LIN {X 0,Y 524.296,Z 355.631,A -85,B 0,C 180,E1 -4781.013,E2 -4781.013} C_VEL
LIN {X 0,Y 524.616,Z 343.771,A -85,B 0,C 180,E1 -4781.889,E2 -4781.889} C_VEL
LIN {X 0,Y 524.905,Z 331.9,A -85,B 0,C 180,E1 -4782.567,E2 -4782.567} C_VEL
LIN {X 0,Y 525.166,Z 319.528,A -85,B 0,C 180,E1 -4783.101,E2 -4783.101} C_VEL
LIN {X 0,Y 525.422,Z 306.835,A -85,B 0,C 180,E1 -4783.489,E2 -4783.489} C_VEL
LIN {X 0,Y 525.58,Z 293.563,A -85,B 0,C 180,E1 -4783.731,E2 -4783.731} C_VEL
LIN {X 0,Y 525.785,Z 203.396,A -85,B 0,C 180,E1 -4784.97,E2 -4784.97} C_VEL
LIN {X 0,Y 524.208,Z 192.625,A -85,B 0,C 180,E1 -4785.178,E2 -4785.178} C_VEL
LIN {X 0,Y 524.604,Z 173.678,A -85,B 0,C 180,E1 -4787.978,E2 -4787.978} C_VEL
LIN {X 0,Y 525.138,Z 150.917,A -85,B 0,C 180,E1 -4791.389,E2 -4791.389} C_VEL
LIN {X 0,Y 525.407,Z 136.058,A -85,B 0,C 180,E1 -4793.659,E2 -4793.659} C_VEL
LIN {X 0,Y 523.975,Z 128.216,A -85,B 0,C 180,E1 -4794.967,E2 -4794.967} C_VEL
LIN {X 0,Y 523.922,Z 128.227,A -85,B 0,C 180,E1 -4798.002,E2 -4798.002} C_VEL
LIN {X 0,Y 523.941,Z 128.22,A -85,B 0,C 180,E1 -4800.854,E2 -4800.854} C_VEL
LIN {X 0,Y 523.962,Z 128.222,A -85,B 0,C 180,E1 -4803.734,E2 -4803.734} C_VEL
LIN {X 0,Y 523.901,Z 128.222,A -85,B 0,C 180,E1 -4806.401,E2 -4806.401} C_VEL
LIN {X 0,Y 523.922,Z 128.22,A -85,B 0,C 180,E1 -4809.085,E2 -4809.085} C_VEL
LIN {X 0,Y 523.942,Z 128.217,A -85,B 0,C 180,E1 -4812.12,E2 -4812.12} C_VEL
LIN {X 0,Y 523.939,Z 128.224,A -85,B 0,C 180,E1 -4815.311,E2 -4815.311} C_VEL
LIN {X 0,Y 523.94,Z 128.218,A -85,B 0,C 180,E1 -4818.692,E2 -4818.692} C_VEL
LIN {X 0,Y 523.914,Z 128.221,A -85,B 0,C 180,E1 -4821.898,E2 -4821.898} C_VEL
LIN {X 0,Y 523.922,Z 128.225,A -85,B 0,C 180,E1 -4824.912,E2 -4824.912} C_VEL
LIN {X 0,Y 523.931,Z 128.219,A -85,B 0,C 180,E1 -4827.681,E2 -4827.681} C_VEL
LIN {X 0,Y 523.935,Z 128.222,A -85,B 0,C 180,E1 -4830.68,E2 -4830.68} C_VEL
LIN {X 0,Y 523.902,Z 128.221,A -85,B 0,C 180,E1 -4833.725,E2 -4833.725} C_VEL
LIN {X 0,Y 523.904,Z 128.223,A -85,B 0,C 180,E1 -4836.269,E2 -4836.269} C_VEL
LIN {X 0,Y 523.928,Z 128.223,A -85,B 0,C 180,E1 -4838.766,E2 -4838.766} C_VEL
LIN {X 0,Y 523.924,Z 128.218,A -85,B 0,C 180,E1 -4841.22,E2 -4841.22} C_VEL
LIN {X 0,Y 523.877,Z 128.224,A -85,B 0,C 180,E1 -4843.637,E2 -4843.637} C_VEL
LIN {X 0,Y 523.959,Z 128.211,A -85,B 0,C 180,E1 -4845.235,E2 -4845.235} C_VEL
LIN {X 0,Y 523.958,Z 128.221,A -85,B 0,C 180,E1 -4848.393,E2 -4848.393} C_VEL
LIN {X 0,Y 523.94,Z 128.214,A -85,B 0,C 180,E1 -4851.515,E2 -4851.515} C_VEL
LIN {X 0,Y 523.997,Z 128.213,A -85,B 0,C 180,E1 -4853.84,E2 -4853.84} C_VEL
LIN {X 0,Y 524.101,Z 128.197,A -85,B 0,C 180,E1 -4857.695,E2 -4857.695} C_VEL
LIN {X 0,Y 524.094,Z 128.204,A -85,B 0,C 180,E1 -4860,E2 -4860} C_VEL
LIN {X 0,Y 524.102,Z 128.195,A -85,B 0,C 180,E1 -4862.306,E2 -4862.306} C_VEL
LIN {X 0,Y 524,Z 128.211,A -85,B 0,C 180,E1 -4866.16,E2 -4866.16} C_VEL
LIN {X 0,Y 523.977,Z 128.212,A -85,B 0,C 180,E1 -4869.262,E2 -4869.262} C_VEL
LIN {X 0,Y 523.997,Z 128.214,A -85,B 0,C 180,E1 -4871.736,E2 -4871.736} C_VEL
LIN {X 0,Y 523.983,Z 128.212,A -85,B 0,C 180,E1 -4875.048,E2 -4875.048} C_VEL
LIN {X 0,Y 523.944,Z 128.216,A -85,B 0,C 180,E1 -4877.97,E2 -4877.97} C_VEL
LIN {X 0,Y 523.958,Z 128.213,A -85,B 0,C 180,E1 -4880.411,E2 -4880.411} C_VEL
LIN {X 0,Y 523.907,Z 128.226,A -85,B 0,C 180,E1 -4882.894,E2 -4882.894} C_VEL
LIN {X 0,Y 523.903,Z 128.224,A -85,B 0,C 180,E1 -4885.421,E2 -4885.421} C_VEL
LIN {X 0,Y 523.92,Z 128.218,A -85,B 0,C 180,E1 -4888.002,E2 -4888.002} C_VEL
LIN {X 0,Y 523.936,Z 128.225,A -85,B 0,C 180,E1 -4890.853,E2 -4890.853} C_VEL
LIN {X 0,Y 523.931,Z 128.217,A -85,B 0,C 180,E1 -4893.73,E2 -4893.73} C_VEL
LIN {X 0,Y 523.905,Z 128.225,A -85,B 0,C 180,E1 -4896.401,E2 -4896.401} C_VEL
LIN {X 0,Y 523.915,Z 128.22,A -85,B 0,C 180,E1 -4899.086,E2 -4899.086} C_VEL
LIN {X 0,Y 523.953,Z 128.214,A -85,B 0,C 180,E1 -4902.119,E2 -4902.119} C_VEL
LIN {X 0,Y 523.946,Z 128.215,A -85,B 0,C 180,E1 -4905.31,E2 -4905.31} C_VEL
LIN {X 0,Y 523.904,Z 128.222,A -85,B 0,C 180,E1 -4906.869,E2 -4906.869} C_VEL
LIN {X 0,Y 523.232,Z 128.305,A -85,B 0,C 180,E1 -4907.51,E2 -4907.51} C_VEL
LIN {X 0,Y 520.37,Z 128.666,A -85,B 0,C 180,E1 -4908.552,E2 -4908.552} C_VEL
LIN {X 0,Y 517.967,Z 128.963,A -85,B 0,C 180,E1 -4909.391,E2 -4909.391} C_VEL
LIN {X 0,Y 516.956,Z 129.093,A -85,B 0,C 180,E1 -4910.039,E2 -4910.039} C_VEL
LIN {X 0,Y 516.885,Z 129.102,A -85,B 0,C 180,E1 -4910.258,E2 -4910.258} C_VEL
LIN {X 0,Y 516.881,Z 129.097,A -85,B 0,C 180,E1 -4913.343,E2 -4913.343} C_VEL
LIN {X 0,Y 516.911,Z 129.099,A -85,B 0,C 180,E1 -4916.121,E2 -4916.121} C_VEL
LIN {X 0,Y 516.896,Z 129.095,A -85,B 0,C 180,E1 -4918.936,E2 -4918.936} C_VEL
LIN {X 0,Y 516.914,Z 129.099,A -85,B 0,C 180,E1 -4921.584,E2 -4921.584} C_VEL
LIN {X 0,Y 516.937,Z 129.095,A -85,B 0,C 180,E1 -4924.211,E2 -4924.211} C_VEL
LIN {X 0,Y 516.978,Z 129.251,A -85,B 0,C 180,E1 -4925.931,E2 -4925.931} C_VEL
LIN {X 0,Y 517.464,Z 133.566,A -85,B 0,C 180,E1 -4926.804,E2 -4926.804} C_VEL
LIN {X 0,Y 517.266,Z 148.39,A -85,B 0,C 180,E1 -4929.687,E2 -4929.687} C_VEL
LIN {X 0,Y 519.159,Z 158.865,A -85,B 0,C 180,E1 -4929.9,E2 -4929.9} C_VEL
LIN {X 0,Y 518.678,Z 255.148,A -85,B 0,C 180,E1 -4931.256,E2 -4931.256} C_VEL
LIN {X 0,Y 518.464,Z 268.883,A -85,B 0,C 180,E1 -4931.617,E2 -4931.617} C_VEL
LIN {X 0,Y 518.279,Z 280.763,A -85,B 0,C 180,E1 -4932.082,E2 -4932.082} C_VEL
LIN {X 0,Y 518.008,Z 293.082,A -85,B 0,C 180,E1 -4932.735,E2 -4932.735} C_VEL
LIN {X 0,Y 517.682,Z 304.709,A -85,B 0,C 180,E1 -4933.536,E2 -4933.536} C_VEL
LIN {X 0,Y 517.386,Z 314.85,A -85,B 0,C 180,E1 -4934.411,E2 -4934.411} C_VEL
LIN {X 0,Y 517.145,Z 324.44,A -85,B 0,C 180,E1 -4935.438,E2 -4935.438} C_VEL
LIN {X 0,Y 516.818,Z 333.435,A -85,B 0,C 180,E1 -4936.633,E2 -4936.633} C_VEL
LIN {X 0,Y 516.649,Z 340.641,A -85,B 0,C 180,E1 -4937.827,E2 -4937.827} C_VEL
LIN {X 0,Y 516.461,Z 346.349,A -85,B 0,C 180,E1 -4939.017,E2 -4939.017} C_VEL
LIN {X 0,Y 516.384,Z 350.822,A -85,B 0,C 180,E1 -4940.204,E2 -4940.204} C_VEL
LIN {X 0,Y 516.348,Z 354.202,A -85,B 0,C 180,E1 -4941.389,E2 -4941.389} C_VEL
LIN {X 0,Y 516.292,Z 357.143,A -85,B 0,C 180,E1 -4942.962,E2 -4942.962} C_VEL
LIN {X 0,Y 516.313,Z 358.016,A -85,B 0,C 180,E1 -4943.748,E2 -4943.748} C_VEL
LIN {X 0,Y 516.309,Z 358.461,A -85,B 0,C 180,E1 -4944.532,E2 -4944.532} C_VEL
LIN {X 0,Y 516.326,Z 358.176,A -85,B 0,C 180,E1 -4946.097,E2 -4946.097} C_VEL
LIN {X 0,Y 516.344,Z 357.465,A -85,B 0,C 180,E1 -4946.878,E2 -4946.878} C_VEL
LIN {X 0,Y 516.267,Z 356.334,A -85,B 0,C 180,E1 -4947.659,E2 -4947.659} C_VEL
LIN {X 0,Y 516.253,Z 352.833,A -85,B 0,C 180,E1 -4949.219,E2 -4949.219} C_VEL
LIN {X 0,Y 516.445,Z 349.035,A -85,B 0,C 180,E1 -4950.389,E2 -4950.389} C_VEL
LIN {X 0,Y 516.44,Z 344.15,A -85,B 0,C 180,E1 -4951.559,E2 -4951.559} C_VEL
LIN {X 0,Y 516.671,Z 338.002,A -85,B 0,C 180,E1 -4952.728,E2 -4952.728} C_VEL
LIN {X 0,Y 516.803,Z 330.352,A -85,B 0,C 180,E1 -4953.898,E2 -4953.898} C_VEL
LIN {X 0,Y 517.111,Z 322.535,A -85,B 0,C 180,E1 -4954.872,E2 -4954.872} C_VEL
LIN {X 0,Y 517.454,Z 311.966,A -85,B 0,C 180,E1 -4955.944,E2 -4955.944} C_VEL
LIN {X 0,Y 517.824,Z 301.13,A -85,B 0,C 180,E1 -4956.82,E2 -4956.82} C_VEL
LIN {X 0,Y 518.163,Z 289.248,A -85,B 0,C 180,E1 -4957.573,E2 -4957.573} C_VEL
LIN {X 0,Y 518.355,Z 277.548,A -85,B 0,C 180,E1 -4958.147,E2 -4958.147} C_VEL
LIN {X 0,Y 518.562,Z 264.854,A -85,B 0,C 180,E1 -4958.597,E2 -4958.597} C_VEL
LIN {X 0,Y 518.631,Z 251.952,A -85,B 0,C 180,E1 -4958.891,E2 -4958.891} C_VEL
LIN {X 0,Y 519.083,Z 157.954,A -85,B 0,C 180,E1 -4960.204,E2 -4960.204} C_VEL
LIN {X 0,Y 517.203,Z 148.275,A -85,B 0,C 180,E1 -4960.421,E2 -4960.421} C_VEL
LIN {X 0,Y 517.436,Z 133.231,A -85,B 0,C 180,E1 -4963.349,E2 -4963.349} C_VEL
LIN {X 0,Y 516.945,Z 129.096,A -85,B 0,C 180,E1 -4964.214,E2 -4964.214} C_VEL
LIN {X 0,Y 516.907,Z 129.094,A -85,B 0,C 180,E1 -4967.404,E2 -4967.404} C_VEL
LIN {X 0,Y 516.94,Z 129.097,A -85,B 0,C 180,E1 -4970.267,E2 -4970.267} C_VEL
LIN {X 0,Y 516.86,Z 129.098,A -85,B 0,C 180,E1 -4973.223,E2 -4973.223} C_VEL
LIN {X 0,Y 516.941,Z 129.095,A -85,B 0,C 180,E1 -4976.195,E2 -4976.195} C_VEL
LIN {X 0,Y 516.919,Z 129.092,A -85,B 0,C 180,E1 -4979.303,E2 -4979.303} C_VEL
LIN {X 0,Y 516.893,Z 129.096,A -85,B 0,C 180,E1 -4982.542,E2 -4982.542} C_VEL
LIN {X 0,Y 516.863,Z 129.101,A -85,B 0,C 180,E1 -4985.328,E2 -4985.328} C_VEL
LIN {X 0,Y 516.876,Z 129.102,A -85,B 0,C 180,E1 -4987.942,E2 -4987.942} C_VEL
LIN {X 0,Y 516.878,Z 129.097,A -85,B 0,C 180,E1 -4990.741,E2 -4990.741} C_VEL
LIN {X 0,Y 516.877,Z 129.098,A -85,B 0,C 180,E1 -4992.83,E2 -4992.83} C_VEL
LIN {X 0,Y 516.889,Z 129.099,A -85,B 0,C 180,E1 -4995.006,E2 -4995.006} C_VEL
LIN {X 0,Y 516.906,Z 129.094,A -85,B 0,C 180,E1 -4998.398,E2 -4998.398} C_VEL
LIN {X 0,Y 516.871,Z 129.104,A -85,B 0,C 180,E1 -5001.283,E2 -5001.283} C_VEL
LIN {X 0,Y 516.862,Z 129.099,A -85,B 0,C 180,E1 -5004.219,E2 -5004.219} C_VEL
LIN {X 0,Y 516.872,Z 129.103,A -85,B 0,C 180,E1 -5007.051,E2 -5007.051} C_VEL
LIN {X 0,Y 516.876,Z 129.098,A -85,B 0,C 180,E1 -5009.795,E2 -5009.795} C_VEL
LIN {X 0,Y 516.91,Z 129.097,A -85,B 0,C 180,E1 -5012.466,E2 -5012.466} C_VEL
LIN {X 0,Y 516.861,Z 129.1,A -85,B 0,C 180,E1 -5015.645,E2 -5015.645} C_VEL
LIN {X 0,Y 516.873,Z 129.103,A -85,B 0,C 180,E1 -5018.461,E2 -5018.461} C_VEL
LIN {X 0,Y 516.878,Z 129.102,A -85,B 0,C 180,E1 -5020.954,E2 -5020.954} C_VEL
LIN {X 0,Y 516.86,Z 129.1,A -85,B 0,C 180,E1 -5023.408,E2 -5023.408} C_VEL
LIN {X 0,Y 516.86,Z 129.101,A -85,B 0,C 180,E1 -5025.833,E2 -5025.833} C_VEL
LIN {X 0,Y 516.935,Z 129.092,A -85,B 0,C 180,E1 -5029.027,E2 -5029.027} C_VEL
LIN {X 0,Y 516.929,Z 129.096,A -85,B 0,C 180,E1 -5032.186,E2 -5032.186} C_VEL
LIN {X 0,Y 516.972,Z 129.09,A -85,B 0,C 180,E1 -5034.539,E2 -5034.539} C_VEL
LIN {X 0,Y 517.061,Z 129.078,A -85,B 0,C 180,E1 -5037.663,E2 -5037.663} C_VEL
LIN {X 0,Y 517.052,Z 129.081,A -85,B 0,C 180,E1 -5040,E2 -5040} C_VEL
LIN {X 0,Y 517.061,Z 129.078,A -85,B 0,C 180,E1 -5042.337,E2 -5042.337} C_VEL
LIN {X 0,Y 516.972,Z 129.089,A -85,B 0,C 180,E1 -5046.244,E2 -5046.244} C_VEL
LIN {X 0,Y 516.923,Z 129.097,A -85,B 0,C 180,E1 -5049.39,E2 -5049.39} C_VEL
LIN {X 0,Y 516.939,Z 129.094,A -85,B 0,C 180,E1 -5051.807,E2 -5051.807} C_VEL
LIN {X 0,Y 516.923,Z 129.096,A -85,B 0,C 180,E1 -5055.143,E2 -5055.143} C_VEL
LIN {X 0,Y 516.899,Z 129.095,A -85,B 0,C 180,E1 -5058.223,E2 -5058.223} C_VEL
LIN {X 0,Y 516.892,Z 129.097,A -85,B 0,C 180,E1 -5060.702,E2 -5060.702} C_VEL
LIN {X 0,Y 516.872,Z 129.098,A -85,B 0,C 180,E1 -5064.074,E2 -5064.074} C_VEL
LIN {X 0,Y 516.896,Z 129.098,A -85,B 0,C 180,E1 -5066.659,E2 -5066.659} C_VEL
LIN {X 0,Y 516.898,Z 129.097,A -85,B 0,C 180,E1 -5069.524,E2 -5069.524} C_VEL
LIN {X 0,Y 516.884,Z 129.1,A -85,B 0,C 180,E1 -5072.544,E2 -5072.544} C_VEL
LIN {X 0,Y 516.856,Z 129.102,A -85,B 0,C 180,E1 -5075.33,E2 -5075.33} C_VEL
LIN {X 0,Y 516.871,Z 129.098,A -85,B 0,C 180,E1 -5077.944,E2 -5077.944} C_VEL
LIN {X 0,Y 516.874,Z 129.103,A -85,B 0,C 180,E1 -5080.743,E2 -5080.743} C_VEL
LIN {X 0,Y 516.875,Z 129.101,A -85,B 0,C 180,E1 -5082.832,E2 -5082.832} C_VEL
LIN {X 0,Y 516.888,Z 129.098,A -85,B 0,C 180,E1 -5085.008,E2 -5085.008} C_VEL
LIN {X 0,Y 516.907,Z 129.1,A -85,B 0,C 180,E1 -5088.4,E2 -5088.4} C_VEL
LIN {X 0,Y 516.876,Z 129.097,A -85,B 0,C 180,E1 -5091.285,E2 -5091.285} C_VEL
LIN {X 0,Y 516.866,Z 129.105,A -85,B 0,C 180,E1 -5094.221,E2 -5094.221} C_VEL
LIN {X 0,Y 516.891,Z 129.095,A -85,B 0,C 180,E1 -5097.054,E2 -5097.054} C_VEL
LIN {X 0,Y 516.889,Z 129.1,A -85,B 0,C 180,E1 -5099.797,E2 -5099.797} C_VEL
LIN {X 0,Y 516.925,Z 129.093,A -85,B 0,C 180,E1 -5102.468,E2 -5102.468} C_VEL
LIN {X 0,Y 516.953,Z 129.223,A -85,B 0,C 180,E1 -5104.941,E2 -5104.941} C_VEL
LIN {X 0,Y 518.403,Z 136.998,A -85,B 0,C 180,E1 -5106.215,E2 -5106.215} C_VEL
LIN {X 0,Y 518.207,Z 149.253,A -85,B 0,C 180,E1 -5108.103,E2 -5108.103} C_VEL
LIN {X 0,Y 517.782,Z 165.52,A -85,B 0,C 180,E1 -5110.578,E2 -5110.578} C_VEL
LIN {X 0,Y 517.435,Z 184.423,A -85,B 0,C 180,E1 -5113.428,E2 -5113.428} C_VEL
LIN {X 0,Y 517.213,Z 192.423,A -85,B 0,C 180,E1 -5114.625,E2 -5114.625} C_VEL
LIN {X 0,Y 519.016,Z 205.194,A -85,B 0,C 180,E1 -5114.86,E2 -5114.86} C_VEL
LIN {X 0,Y 518.594,Z 301.016,A -85,B 0,C 180,E1 -5116.207,E2 -5116.207} C_VEL
LIN {X 0,Y 518.375,Z 313.548,A -85,B 0,C 180,E1 -5116.526,E2 -5116.526} C_VEL
LIN {X 0,Y 518.073,Z 326.498,A -85,B 0,C 180,E1 -5117.017,E2 -5117.017} C_VEL
LIN {X 0,Y 517.775,Z 338.996,A -85,B 0,C 180,E1 -5117.669,E2 -5117.669} C_VEL
LIN {X 0,Y 517.478,Z 350.426,A -85,B 0,C 180,E1 -5118.445,E2 -5118.445} C_VEL
LIN {X 0,Y 517.194,Z 360.897,A -85,B 0,C 180,E1 -5119.331,E2 -5119.331} C_VEL
LIN {X 0,Y 516.905,Z 369.459,A -85,B 0,C 180,E1 -5120.216,E2 -5120.216} C_VEL
LIN {X 0,Y 516.68,Z 377.362,A -85,B 0,C 180,E1 -5121.199,E2 -5121.199} C_VEL
LIN {X 0,Y 516.515,Z 385.085,A -85,B 0,C 180,E1 -5122.377,E2 -5122.377} C_VEL
LIN {X 0,Y 516.373,Z 392.205,A -85,B 0,C 180,E1 -5123.75,E2 -5123.75} C_VEL
LIN {X 0,Y 516.312,Z 396.943,A -85,B 0,C 180,E1 -5124.925,E2 -5124.925} C_VEL
LIN {X 0,Y 516.351,Z 400.566,A -85,B 0,C 180,E1 -5126.099,E2 -5126.099} C_VEL
LIN {X 0,Y 516.303,Z 402.432,A -85,B 0,C 180,E1 -5126.88,E2 -5126.88} C_VEL
LIN {X 0,Y 516.264,Z 403.831,A -85,B 0,C 180,E1 -5127.66,E2 -5127.66} C_VEL
LIN {X 0,Y 516.172,Z 405.435,A -85,B 0,C 180,E1 -5129.221,E2 -5129.221} C_VEL
LIN {X 0,Y 516.173,Z 405.651,A -85,B 0,C 180,E1 -5130.001,E2 -5130.001} C_VEL
LIN {X 0,Y 516.193,Z 404.822,A -85,B 0,C 180,E1 -5131.561,E2 -5131.561} C_VEL
LIN {X 0,Y 516.264,Z 403.825,A -85,B 0,C 180,E1 -5132.341,E2 -5132.341} C_VEL
LIN {X 0,Y 516.303,Z 402.425,A -85,B 0,C 180,E1 -5133.122,E2 -5133.122} C_VEL
LIN {X 0,Y 516.31,Z 399.476,A -85,B 0,C 180,E1 -5134.294,E2 -5134.294} C_VEL
LIN {X 0,Y 516.367,Z 395.487,A -85,B 0,C 180,E1 -5135.468,E2 -5135.468} C_VEL
LIN {X 0,Y 516.427,Z 389.342,A -85,B 0,C 180,E1 -5136.841,E2 -5136.841} C_VEL
LIN {X 0,Y 516.568,Z 382.649,A -85,B 0,C 180,E1 -5138.017,E2 -5138.017} C_VEL
LIN {X 0,Y 516.756,Z 374.336,A -85,B 0,C 180,E1 -5139.196,E2 -5139.196} C_VEL
LIN {X 0,Y 516.985,Z 365.819,A -85,B 0,C 180,E1 -5140.18,E2 -5140.18} C_VEL
LIN {X 0,Y 517.302,Z 355.3,A -85,B 0,C 180,E1 -5141.163,E2 -5141.163} C_VEL
LIN {X 0,Y 517.623,Z 343.438,A -85,B 0,C 180,E1 -5142.052,E2 -5142.052} C_VEL
LIN {X 0,Y 517.941,Z 331.566,A -85,B 0,C 180,E1 -5142.739,E2 -5142.739} C_VEL
LIN {X 0,Y 518.227,Z 319.193,A -85,B 0,C 180,E1 -5143.28,E2 -5143.28} C_VEL
LIN {X 0,Y 518.506,Z 306.499,A -85,B 0,C 180,E1 -5143.672,E2 -5143.672} C_VEL
LIN {X 0,Y 518.675,Z 291.432,A -85,B 0,C 180,E1 -5143.942,E2 -5143.942} C_VEL
LIN {X 0,Y 518.91,Z 204.051,A -85,B 0,C 180,E1 -5145.159,E2 -5145.159} C_VEL
LIN {X 0,Y 517.223,Z 192.309,A -85,B 0,C 180,E1 -5145.386,E2 -5145.386} C_VEL
LIN {X 0,Y 517.725,Z 170.878,A -85,B 0,C 180,E1 -5148.603,E2 -5148.603} C_VEL
LIN {X 0,Y 518.192,Z 152,A -85,B 0,C 180,E1 -5151.481,E2 -5151.481} C_VEL
LIN {X 0,Y 518.466,Z 137.166,A -85,B 0,C 180,E1 -5153.783,E2 -5153.783} C_VEL
LIN {X 0,Y 516.916,Z 129.095,A -85,B 0,C 180,E1 -5155.143,E2 -5155.143} C_VEL
LIN {X 0,Y 516.886,Z 129.103,A -85,B 0,C 180,E1 -5157.896,E2 -5157.896} C_VEL
LIN {X 0,Y 516.889,Z 129.104,A -85,B 0,C 180,E1 -5160.204,E2 -5160.204} C_VEL
LIN {X 0,Y 516.898,Z 129.096,A -85,B 0,C 180,E1 -5162.947,E2 -5162.947} C_VEL
LIN {X 0,Y 516.87,Z 129.105,A -85,B 0,C 180,E1 -5165.781,E2 -5165.781} C_VEL
LIN {X 0,Y 516.882,Z 129.095,A -85,B 0,C 180,E1 -5168.716,E2 -5168.716} C_VEL
LIN {X 0,Y 516.907,Z 129.097,A -85,B 0,C 180,E1 -5171.776,E2 -5171.776} C_VEL
LIN {X 0,Y 516.897,Z 129.097,A -85,B 0,C 180,E1 -5175.007,E2 -5175.007} C_VEL
LIN {X 0,Y 516.903,Z 129.093,A -85,B 0,C 180,E1 -5178.4,E2 -5178.4} C_VEL
LIN {X 0,Y 516.877,Z 129.104,A -85,B 0,C 180,E1 -5181.284,E2 -5181.284} C_VEL
LIN {X 0,Y 516.868,Z 129.098,A -85,B 0,C 180,E1 -5184.219,E2 -5184.219} C_VEL
LIN {X 0,Y 516.88,Z 129.104,A -85,B 0,C 180,E1 -5187.052,E2 -5187.052} C_VEL
LIN {X 0,Y 516.862,Z 129.098,A -85,B 0,C 180,E1 -5189.794,E2 -5189.794} C_VEL
LIN {X 0,Y 516.874,Z 129.099,A -85,B 0,C 180,E1 -5192.464,E2 -5192.464} C_VEL
LIN {X 0,Y 516.844,Z 129.105,A -85,B 0,C 180,E1 -5195.068,E2 -5195.068} C_VEL
LIN {X 0,Y 516.869,Z 129.097,A -85,B 0,C 180,E1 -5197.622,E2 -5197.622} C_VEL
LIN {X 0,Y 516.913,Z 129.092,A -85,B 0,C 180,E1 -5200.129,E2 -5200.129} C_VEL
LIN {X 0,Y 516.877,Z 129.103,A -85,B 0,C 180,E1 -5202.594,E2 -5202.594} C_VEL
LIN {X 0,Y 516.929,Z 129.088,A -85,B 0,C 180,E1 -5205.03,E2 -5205.03} C_VEL
LIN {X 0,Y 516.918,Z 129.098,A -85,B 0,C 180,E1 -5208.233,E2 -5208.233} C_VEL
LIN {X 0,Y 516.914,Z 129.088,A -85,B 0,C 180,E1 -5211.399,E2 -5211.399} C_VEL
LIN {X 0,Y 516.975,Z 129.086,A -85,B 0,C 180,E1 -5214.539,E2 -5214.539} C_VEL
LIN {X 0,Y 517.07,Z 129.073,A -85,B 0,C 180,E1 -5217.663,E2 -5217.663} C_VEL
LIN {X 0,Y 517.063,Z 129.08,A -85,B 0,C 180,E1 -5220,E2 -5220} C_VEL
LIN {X 0,Y 517.071,Z 129.07,A -85,B 0,C 180,E1 -5222.337,E2 -5222.337} C_VEL
LIN {X 0,Y 516.967,Z 129.086,A -85,B 0,C 180,E1 -5226.244,E2 -5226.244} C_VEL
LIN {X 0,Y 516.934,Z 129.091,A -85,B 0,C 180,E1 -5229.39,E2 -5229.39} C_VEL
LIN {X 0,Y 516.952,Z 129.091,A -85,B 0,C 180,E1 -5231.807,E2 -5231.807} C_VEL
LIN {X 0,Y 516.936,Z 129.091,A -85,B 0,C 180,E1 -5235.143,E2 -5235.143} C_VEL
LIN {X 0,Y 516.911,Z 129.091,A -85,B 0,C 180,E1 -5238.223,E2 -5238.223} C_VEL
LIN {X 0,Y 516.905,Z 129.093,A -85,B 0,C 180,E1 -5240.702,E2 -5240.702} C_VEL
LIN {X 0,Y 516.885,Z 129.093,A -85,B 0,C 180,E1 -5244.074,E2 -5244.074} C_VEL
LIN {X 0,Y 516.895,Z 129.098,A -85,B 0,C 180,E1 -5246.66,E2 -5246.66} C_VEL
LIN {X 0,Y 516.908,Z 129.093,A -85,B 0,C 180,E1 -5249.523,E2 -5249.523} C_VEL
LIN {X 0,Y 516.895,Z 129.099,A -85,B 0,C 180,E1 -5252.543,E2 -5252.543} C_VEL
LIN {X 0,Y 516.867,Z 129.098,A -85,B 0,C 180,E1 -5255.33,E2 -5255.33} C_VEL
LIN {X 0,Y 516.881,Z 129.096,A -85,B 0,C 180,E1 -5257.943,E2 -5257.943} C_VEL
LIN {X 0,Y 516.885,Z 129.094,A -85,B 0,C 180,E1 -5260.742,E2 -5260.742} C_VEL
LIN {X 0,Y 516.885,Z 129.098,A -85,B 0,C 180,E1 -5262.832,E2 -5262.832} C_VEL
LIN {X 0,Y 516.898,Z 129.094,A -85,B 0,C 180,E1 -5265.007,E2 -5265.007} C_VEL
LIN {X 0,Y 516.913,Z 129.098,A -85,B 0,C 180,E1 -5268.399,E2 -5268.399} C_VEL
LIN {X 0,Y 516.885,Z 129.102,A -85,B 0,C 180,E1 -5270.258,E2 -5270.258} C_VEL
LIN {X 0,Y 516.249,Z 129.188,A -85,B 0,C 180,E1 -5270.908,E2 -5270.908} C_VEL
LIN {X 0,Y 513.406,Z 129.544,A -85,B 0,C 180,E1 -5271.963,E2 -5271.963} C_VEL
LIN {X 0,Y 510.976,Z 129.841,A -85,B 0,C 180,E1 -5272.813,E2 -5272.813} C_VEL
LIN {X 0,Y 509.918,Z 129.968,A -85,B 0,C 180,E1 -5273.47,E2 -5273.47} C_VEL
LIN {X 0,Y 509.826,Z 129.978,A -85,B 0,C 180,E1 -5273.692,E2 -5273.692} C_VEL
LIN {X 0,Y 509.863,Z 129.972,A -85,B 0,C 180,E1 -5276.539,E2 -5276.539} C_VEL
LIN {X 0,Y 509.85,Z 129.974,A -85,B 0,C 180,E1 -5279.334,E2 -5279.334} C_VEL
LIN {X 0,Y 509.888,Z 129.974,A -85,B 0,C 180,E1 -5282.054,E2 -5282.054} C_VEL
LIN {X 0,Y 509.884,Z 129.971,A -85,B 0,C 180,E1 -5284.704,E2 -5284.704} C_VEL
LIN {X 0,Y 509.925,Z 130.125,A -85,B 0,C 180,E1 -5285.793,E2 -5285.793} C_VEL
LIN {X 0,Y 510.486,Z 134.461,A -85,B 0,C 180,E1 -5286.683,E2 -5286.683} C_VEL
LIN {X 0,Y 510.303,Z 148.728,A -85,B 0,C 180,E1 -5289.474,E2 -5289.474} C_VEL
LIN {X 0,Y 512.299,Z 159.889,A -85,B 0,C 180,E1 -5289.7,E2 -5289.7} C_VEL
LIN {X 0,Y 511.813,Z 255.635,A -85,B 0,C 180,E1 -5291.07,E2 -5291.07} C_VEL
LIN {X 0,Y 511.577,Z 269.311,A -85,B 0,C 180,E1 -5291.435,E2 -5291.435} C_VEL
LIN {X 0,Y 511.364,Z 281.795,A -85,B 0,C 180,E1 -5291.935,E2 -5291.935} C_VEL
LIN {X 0,Y 511.067,Z 293.899,A -85,B 0,C 180,E1 -5292.596,E2 -5292.596} C_VEL
LIN {X 0,Y 510.713,Z 305.43,A -85,B 0,C 180,E1 -5293.408,E2 -5293.408} C_VEL
LIN {X 0,Y 510.407,Z 315.709,A -85,B 0,C 180,E1 -5294.316,E2 -5294.316} C_VEL
LIN {X 0,Y 510.161,Z 324.192,A -85,B 0,C 180,E1 -5295.234,E2 -5295.234} C_VEL
LIN {X 0,Y 509.834,Z 333.285,A -85,B 0,C 180,E1 -5296.447,E2 -5296.447} C_VEL
LIN {X 0,Y 509.607,Z 340.58,A -85,B 0,C 180,E1 -5297.657,E2 -5297.657} C_VEL
LIN {X 0,Y 509.432,Z 346.385,A -85,B 0,C 180,E1 -5298.863,E2 -5298.863} C_VEL
LIN {X 0,Y 509.314,Z 350.928,A -85,B 0,C 180,E1 -5300.067,E2 -5300.067} C_VEL
LIN {X 0,Y 509.255,Z 354.367,A -85,B 0,C 180,E1 -5301.268,E2 -5301.268} C_VEL
LIN {X 0,Y 509.238,Z 356.072,A -85,B 0,C 180,E1 -5302.067,E2 -5302.067} C_VEL
LIN {X 0,Y 509.262,Z 358.271,A -85,B 0,C 180,E1 -5303.661,E2 -5303.661} C_VEL
LIN {X 0,Y 509.241,Z 358.769,A -85,B 0,C 180,E1 -5304.456,E2 -5304.456} C_VEL
LIN {X 0,Y 509.148,Z 358.849,A -85,B 0,C 180,E1 -5305.249,E2 -5305.249} C_VEL
LIN {X 0,Y 509.251,Z 358.54,A -85,B 0,C 180,E1 -5306.043,E2 -5306.043} C_VEL
LIN {X 0,Y 509.254,Z 357.857,A -85,B 0,C 180,E1 -5306.835,E2 -5306.835} C_VEL
LIN {X 0,Y 509.197,Z 356.78,A -85,B 0,C 180,E1 -5307.626,E2 -5307.626} C_VEL
LIN {X 0,Y 509.165,Z 353.339,A -85,B 0,C 180,E1 -5309.208,E2 -5309.208} C_VEL
LIN {X 0,Y 509.361,Z 349.602,A -85,B 0,C 180,E1 -5310.395,E2 -5310.395} C_VEL
LIN {X 0,Y 509.372,Z 344.783,A -85,B 0,C 180,E1 -5311.581,E2 -5311.581} C_VEL
LIN {X 0,Y 509.618,Z 338.707,A -85,B 0,C 180,E1 -5312.766,E2 -5312.766} C_VEL
LIN {X 0,Y 509.769,Z 331.179,A -85,B 0,C 180,E1 -5313.952,E2 -5313.952} C_VEL
LIN {X 0,Y 510.088,Z 323.467,A -85,B 0,C 180,E1 -5314.939,E2 -5314.939} C_VEL
LIN {X 0,Y 510.464,Z 313.019,A -85,B 0,C 180,E1 -5316.025,E2 -5316.025} C_VEL
LIN {X 0,Y 510.87,Z 302.385,A -85,B 0,C 180,E1 -5316.913,E2 -5316.913} C_VEL
LIN {X 0,Y 511.159,Z 292.061,A -85,B 0,C 180,E1 -5317.604,E2 -5317.604} C_VEL
LIN {X 0,Y 511.421,Z 279.584,A -85,B 0,C 180,E1 -5318.25,E2 -5318.25} C_VEL
LIN {X 0,Y 511.638,Z 266.618,A -85,B 0,C 180,E1 -5318.74,E2 -5318.74} C_VEL
LIN {X 0,Y 511.77,Z 253.36,A -85,B 0,C 180,E1 -5319.061,E2 -5319.061} C_VEL
LIN {X 0,Y 512.238,Z 158.595,A -85,B 0,C 180,E1 -5320.405,E2 -5320.405} C_VEL
LIN {X 0,Y 510.236,Z 148.618,A -85,B 0,C 180,E1 -5320.615,E2 -5320.615} C_VEL
LIN {X 0,Y 510.467,Z 134.725,A -85,B 0,C 180,E1 -5323.332,E2 -5323.332} C_VEL
LIN {X 0,Y 509.919,Z 129.971,A -85,B 0,C 180,E1 -5324.312,E2 -5324.312} C_VEL
LIN {X 0,Y 509.879,Z 129.971,A -85,B 0,C 180,E1 -5327.651,E2 -5327.651} C_VEL
LIN {X 0,Y 509.887,Z 129.973,A -85,B 0,C 180,E1 -5330.4,E2 -5330.4} C_VEL
LIN {X 0,Y 509.822,Z 129.977,A -85,B 0,C 180,E1 -5333.563,E2 -5333.563} C_VEL
LIN {X 0,Y 509.909,Z 129.969,A -85,B 0,C 180,E1 -5336.377,E2 -5336.377} C_VEL
LIN {X 0,Y 509.87,Z 129.97,A -85,B 0,C 180,E1 -5338.843,E2 -5338.843} C_VEL
LIN {X 0,Y 509.818,Z 129.98,A -85,B 0,C 180,E1 -5341.589,E2 -5341.589} C_VEL
LIN {X 0,Y 509.844,Z 129.974,A -85,B 0,C 180,E1 -5344.413,E2 -5344.413} C_VEL
LIN {X 0,Y 509.813,Z 129.98,A -85,B 0,C 180,E1 -5347.34,E2 -5347.34} C_VEL
LIN {X 0,Y 509.833,Z 129.975,A -85,B 0,C 180,E1 -5350.381,E2 -5350.381} C_VEL
LIN {X 0,Y 509.817,Z 129.979,A -85,B 0,C 180,E1 -5353.061,E2 -5353.061} C_VEL
LIN {X 0,Y 509.816,Z 129.981,A -85,B 0,C 180,E1 -5355.792,E2 -5355.792} C_VEL
LIN {X 0,Y 509.848,Z 129.974,A -85,B 0,C 180,E1 -5358.573,E2 -5358.573} C_VEL
LIN {X 0,Y 509.842,Z 129.976,A -85,B 0,C 180,E1 -5361.786,E2 -5361.786} C_VEL
LIN {X 0,Y 509.82,Z 129.979,A -85,B 0,C 180,E1 -5364.621,E2 -5364.621} C_VEL
LIN {X 0,Y 509.85,Z 129.976,A -85,B 0,C 180,E1 -5367.48,E2 -5367.48} C_VEL
LIN {X 0,Y 509.848,Z 129.974,A -85,B 0,C 180,E1 -5370.273,E2 -5370.273} C_VEL
LIN {X 0,Y 509.861,Z 129.977,A -85,B 0,C 180,E1 -5372.943,E2 -5372.943} C_VEL
LIN {X 0,Y 509.806,Z 129.982,A -85,B 0,C 180,E1 -5376.435,E2 -5376.435} C_VEL
LIN {X 0,Y 509.903,Z 129.967,A -85,B 0,C 180,E1 -5379.844,E2 -5379.844} C_VEL
LIN {X 0,Y 509.833,Z 129.977,A -85,B 0,C 180,E1 -5383.173,E2 -5383.173} C_VEL
LIN {X 0,Y 509.833,Z 129.976,A -85,B 0,C 180,E1 -5385.633,E2 -5385.633} C_VEL
LIN {X 0,Y 509.898,Z 129.97,A -85,B 0,C 180,E1 -5388.874,E2 -5388.874} C_VEL
LIN {X 0,Y 509.894,Z 129.972,A -85,B 0,C 180,E1 -5392.077,E2 -5392.077} C_VEL
LIN {X 0,Y 509.926,Z 129.968,A -85,B 0,C 180,E1 -5394.464,E2 -5394.464} C_VEL
LIN {X 0,Y 510.029,Z 129.954,A -85,B 0,C 180,E1 -5397.631,E2 -5397.631} C_VEL
LIN {X 0,Y 510.021,Z 129.956,A -85,B 0,C 180,E1 -5400,E2 -5400} C_VEL
LIN {X 0,Y 510.03,Z 129.954,A -85,B 0,C 180,E1 -5402.369,E2 -5402.369} C_VEL
LIN {X 0,Y 509.934,Z 129.968,A -85,B 0,C 180,E1 -5405.536,E2 -5405.536} C_VEL
LIN {X 0,Y 509.887,Z 129.969,A -85,B 0,C 180,E1 -5408.721,E2 -5408.721} C_VEL
LIN {X 0,Y 509.891,Z 129.972,A -85,B 0,C 180,E1 -5411.932,E2 -5411.932} C_VEL
LIN {X 0,Y 509.882,Z 129.975,A -85,B 0,C 180,E1 -5415.242,E2 -5415.242} C_VEL
LIN {X 0,Y 509.844,Z 129.974,A -85,B 0,C 180,E1 -5418.484,E2 -5418.484} C_VEL
LIN {X 0,Y 509.834,Z 129.98,A -85,B 0,C 180,E1 -5421.002,E2 -5421.002} C_VEL
LIN {X 0,Y 509.806,Z 129.982,A -85,B 0,C 180,E1 -5423.565,E2 -5423.565} C_VEL
LIN {X 0,Y 509.863,Z 129.977,A -85,B 0,C 180,E1 -5427.057,E2 -5427.057} C_VEL
LIN {X 0,Y 509.846,Z 129.974,A -85,B 0,C 180,E1 -5429.752,E2 -5429.752} C_VEL
LIN {X 0,Y 509.857,Z 129.979,A -85,B 0,C 180,E1 -5432.774,E2 -5432.774} C_VEL
LIN {X 0,Y 509.816,Z 129.977,A -85,B 0,C 180,E1 -5435.579,E2 -5435.579} C_VEL
LIN {X 0,Y 509.841,Z 129.977,A -85,B 0,C 180,E1 -5438.339,E2 -5438.339} C_VEL
LIN {X 0,Y 509.847,Z 129.973,A -85,B 0,C 180,E1 -5441.427,E2 -5441.427} C_VEL
LIN {X 0,Y 509.832,Z 129.979,A -85,B 0,C 180,E1 -5444.671,E2 -5444.671} C_VEL
LIN {X 0,Y 509.826,Z 129.975,A -85,B 0,C 180,E1 -5447.511,E2 -5447.511} C_VEL
LIN {X 0,Y 509.841,Z 129.977,A -85,B 0,C 180,E1 -5450.649,E2 -5450.649} C_VEL
LIN {X 0,Y 509.82,Z 129.977,A -85,B 0,C 180,E1 -5453.648,E2 -5453.648} C_VEL
LIN {X 0,Y 509.855,Z 129.974,A -85,B 0,C 180,E1 -5456.54,E2 -5456.54} C_VEL
LIN {X 0,Y 509.842,Z 129.973,A -85,B 0,C 180,E1 -5459.335,E2 -5459.335} C_VEL
LIN {X 0,Y 509.889,Z 129.974,A -85,B 0,C 180,E1 -5462.056,E2 -5462.056} C_VEL
LIN {X 0,Y 509.899,Z 130.093,A -85,B 0,C 180,E1 -5464.777,E2 -5464.777} C_VEL
LIN {X 0,Y 511.517,Z 139.324,A -85,B 0,C 180,E1 -5466.305,E2 -5466.305} C_VEL
LIN {X 0,Y 511.029,Z 159.092,A -85,B 0,C 180,E1 -5469.372,E2 -5469.372} C_VEL
LIN {X 0,Y 510.548,Z 178.684,A -85,B 0,C 180,E1 -5472.373,E2 -5472.373} C_VEL
LIN {X 0,Y 510.21,Z 192.104,A -85,B 0,C 180,E1 -5474.41,E2 -5474.41} C_VEL
LIN {X 0,Y 512.195,Z 206.958,A -85,B 0,C 180,E1 -5474.683,E2 -5474.683} C_VEL
LIN {X 0,Y 511.707,Z 300.687,A -85,B 0,C 180,E1 -5476.018,E2 -5476.018} C_VEL
LIN {X 0,Y 511.476,Z 313.222,A -85,B 0,C 180,E1 -5476.341,E2 -5476.341} C_VEL
LIN {X 0,Y 511.129,Z 326.171,A -85,B 0,C 180,E1 -5476.837,E2 -5476.837} C_VEL
LIN {X 0,Y 510.822,Z 337.797,A -85,B 0,C 180,E1 -5477.444,E2 -5477.444} C_VEL
LIN {X 0,Y 510.473,Z 348.8,A -85,B 0,C 180,E1 -5478.184,E2 -5478.184} C_VEL
LIN {X 0,Y 510.226,Z 359.497,A -85,B 0,C 180,E1 -5479.083,E2 -5479.083} C_VEL
LIN {X 0,Y 509.849,Z 369.133,A -85,B 0,C 180,E1 -5480.079,E2 -5480.079} C_VEL
LIN {X 0,Y 509.639,Z 377.038,A -85,B 0,C 180,E1 -5481.076,E2 -5481.076} C_VEL
LIN {X 0,Y 509.427,Z 384.76,A -85,B 0,C 180,E1 -5482.271,E2 -5482.271} C_VEL
LIN {X 0,Y 509.287,Z 391.881,A -85,B 0,C 180,E1 -5483.663,E2 -5483.663} C_VEL
LIN {X 0,Y 509.241,Z 396.62,A -85,B 0,C 180,E1 -5484.854,E2 -5484.854} C_VEL
LIN {X 0,Y 509.245,Z 400.243,A -85,B 0,C 180,E1 -5486.044,E2 -5486.044} C_VEL
LIN {X 0,Y 509.219,Z 402.109,A -85,B 0,C 180,E1 -5486.836,E2 -5486.836} C_VEL
LIN {X 0,Y 509.193,Z 403.509,A -85,B 0,C 180,E1 -5487.628,E2 -5487.628} C_VEL
LIN {X 0,Y 509.084,Z 405.112,A -85,B 0,C 180,E1 -5489.21,E2 -5489.21} C_VEL
LIN {X 0,Y 509.083,Z 405.327,A -85,B 0,C 180,E1 -5490.001,E2 -5490.001} C_VEL
LIN {X 0,Y 509.113,Z 404.499,A -85,B 0,C 180,E1 -5491.583,E2 -5491.583} C_VEL
LIN {X 0,Y 509.193,Z 403.502,A -85,B 0,C 180,E1 -5492.374,E2 -5492.374} C_VEL
LIN {X 0,Y 509.219,Z 402.1,A -85,B 0,C 180,E1 -5493.165,E2 -5493.165} C_VEL
LIN {X 0,Y 509.203,Z 399.149,A -85,B 0,C 180,E1 -5494.354,E2 -5494.354} C_VEL
LIN {X 0,Y 509.278,Z 395.159,A -85,B 0,C 180,E1 -5495.544,E2 -5495.544} C_VEL
LIN {X 0,Y 509.344,Z 389.124,A -85,B 0,C 180,E1 -5496.915,E2 -5496.915} C_VEL
LIN {X 0,Y 509.494,Z 382.32,A -85,B 0,C 180,E1 -5498.129,E2 -5498.129} C_VEL
LIN {X 0,Y 509.716,Z 374.006,A -85,B 0,C 180,E1 -5499.324,E2 -5499.324} C_VEL
LIN {X 0,Y 509.958,Z 365.488,A -85,B 0,C 180,E1 -5500.321,E2 -5500.321} C_VEL
LIN {X 0,Y 510.3,Z 354.969,A -85,B 0,C 180,E1 -5501.319,E2 -5501.319} C_VEL
LIN {X 0,Y 510.618,Z 343.97,A -85,B 0,C 180,E1 -5502.159,E2 -5502.159} C_VEL
LIN {X 0,Y 510.939,Z 333.164,A -85,B 0,C 180,E1 -5502.815,E2 -5502.815} C_VEL
LIN {X 0,Y 511.278,Z 321.469,A -85,B 0,C 180,E1 -5503.363,E2 -5503.363} C_VEL
LIN {X 0,Y 511.563,Z 308.913,A -85,B 0,C 180,E1 -5503.785,E2 -5503.785} C_VEL
LIN {X 0,Y 511.781,Z 296.2,A -85,B 0,C 180,E1 -5504.058,E2 -5504.058} C_VEL
LIN {X 0,Y 512.004,Z 204.435,A -85,B 0,C 180,E1 -5505.359,E2 -5505.359} C_VEL
LIN {X 0,Y 510.205,Z 191.957,A -85,B 0,C 180,E1 -5505.608,E2 -5505.608} C_VEL
LIN {X 0,Y 510.728,Z 171.948,A -85,B 0,C 180,E1 -5508.66,E2 -5508.66} C_VEL
LIN {X 0,Y 511.246,Z 153.102,A -85,B 0,C 180,E1 -5511.576,E2 -5511.576} C_VEL
LIN {X 0,Y 511.511,Z 138.288,A -85,B 0,C 180,E1 -5513.912,E2 -5513.912} C_VEL
LIN {X 0,Y 509.86,Z 129.974,A -85,B 0,C 180,E1 -5515.352,E2 -5515.352} C_VEL
LIN {X 0,Y 509.837,Z 129.982,A -85,B 0,C 180,E1 -5518.088,E2 -5518.088} C_VEL
LIN {X 0,Y 509.845,Z 129.977,A -85,B 0,C 180,E1 -5520.666,E2 -5520.666} C_VEL
LIN {X 0,Y 509.861,Z 129.976,A -85,B 0,C 180,E1 -5523.461,E2 -5523.461} C_VEL
LIN {X 0,Y 509.811,Z 129.977,A -85,B 0,C 180,E1 -5526.355,E2 -5526.355} C_VEL
LIN {X 0,Y 509.848,Z 129.976,A -85,B 0,C 180,E1 -5529.353,E2 -5529.353} C_VEL
LIN {X 0,Y 509.817,Z 129.975,A -85,B 0,C 180,E1 -5532.492,E2 -5532.492} C_VEL
LIN {X 0,Y 509.84,Z 129.98,A -85,B 0,C 180,E1 -5535.33,E2 -5535.33} C_VEL
LIN {X 0,Y 509.845,Z 129.973,A -85,B 0,C 180,E1 -5538.573,E2 -5538.573} C_VEL
LIN {X 0,Y 509.85,Z 129.974,A -85,B 0,C 180,E1 -5541.787,E2 -5541.787} C_VEL
LIN {X 0,Y 509.827,Z 129.977,A -85,B 0,C 180,E1 -5544.622,E2 -5544.622} C_VEL
LIN {X 0,Y 509.858,Z 129.974,A -85,B 0,C 180,E1 -5547.481,E2 -5547.481} C_VEL
LIN {X 0,Y 509.852,Z 129.972,A -85,B 0,C 180,E1 -5550.275,E2 -5550.275} C_VEL
LIN {X 0,Y 509.824,Z 129.982,A -85,B 0,C 180,E1 -5552.941,E2 -5552.941} C_VEL
LIN {X 0,Y 509.834,Z 129.974,A -85,B 0,C 180,E1 -5555.572,E2 -5555.572} C_VEL
LIN {X 0,Y 509.813,Z 129.978,A -85,B 0,C 180,E1 -5558.148,E2 -5558.148} C_VEL
LIN {X 0,Y 509.842,Z 129.977,A -85,B 0,C 180,E1 -5560.681,E2 -5560.681} C_VEL
LIN {X 0,Y 509.794,Z 129.979,A -85,B 0,C 180,E1 -5563.172,E2 -5563.172} C_VEL
LIN {X 0,Y 509.839,Z 129.97,A -85,B 0,C 180,E1 -5565.633,E2 -5565.633} C_VEL
LIN {X 0,Y 509.858,Z 129.972,A -85,B 0,C 180,E1 -5568.873,E2 -5568.873} C_VEL
LIN {X 0,Y 509.872,Z 129.972,A -85,B 0,C 180,E1 -5572.077,E2 -5572.077} C_VEL
LIN {X 0,Y 509.931,Z 129.965,A -85,B 0,C 180,E1 -5574.464,E2 -5574.464} C_VEL
LIN {X 0,Y 510.038,Z 129.948,A -85,B 0,C 180,E1 -5577.631,E2 -5577.631} C_VEL
LIN {X 0,Y 510.032,Z 129.956,A -85,B 0,C 180,E1 -5580,E2 -5580} C_VEL
LIN {X 0,Y 510.04,Z 129.946,A -85,B 0,C 180,E1 -5582.369,E2 -5582.369} C_VEL
LIN {X 0,Y 509.935,Z 129.966,A -85,B 0,C 180,E1 -5585.536,E2 -5585.536} C_VEL
LIN {X 0,Y 509.898,Z 129.961,A -85,B 0,C 180,E1 -5588.721,E2 -5588.721} C_VEL
LIN {X 0,Y 509.904,Z 129.967,A -85,B 0,C 180,E1 -5591.932,E2 -5591.932} C_VEL
LIN {X 0,Y 509.895,Z 129.969,A -85,B 0,C 180,E1 -5595.242,E2 -5595.242} C_VEL
LIN {X 0,Y 509.856,Z 129.97,A -85,B 0,C 180,E1 -5598.484,E2 -5598.484} C_VEL
LIN {X 0,Y 509.846,Z 129.976,A -85,B 0,C 180,E1 -5601.002,E2 -5601.002} C_VEL
LIN {X 0,Y 509.818,Z 129.975,A -85,B 0,C 180,E1 -5603.564,E2 -5603.564} C_VEL
LIN {X 0,Y 509.874,Z 129.97,A -85,B 0,C 180,E1 -5606.37,E2 -5606.37} C_VEL
LIN {X 0,Y 509.852,Z 129.977,A -85,B 0,C 180,E1 -5608.846,E2 -5608.846} C_VEL
LIN {X 0,Y 509.819,Z 129.975,A -85,B 0,C 180,E1 -5611.591,E2 -5611.591} C_VEL
LIN {X 0,Y 509.84,Z 129.977,A -85,B 0,C 180,E1 -5614.415,E2 -5614.415} C_VEL
LIN {X 0,Y 509.818,Z 129.976,A -85,B 0,C 180,E1 -5617.341,E2 -5617.341} C_VEL
LIN {X 0,Y 509.84,Z 129.975,A -85,B 0,C 180,E1 -5620.382,E2 -5620.382} C_VEL
LIN {X 0,Y 509.825,Z 129.976,A -85,B 0,C 180,E1 -5623.062,E2 -5623.062} C_VEL
LIN {X 0,Y 509.825,Z 129.976,A -85,B 0,C 180,E1 -5625.794,E2 -5625.794} C_VEL
LIN {X 0,Y 509.856,Z 129.975,A -85,B 0,C 180,E1 -5628.574,E2 -5628.574} C_VEL
LIN {X 0,Y 509.855,Z 129.975,A -85,B 0,C 180,E1 -5631.787,E2 -5631.787} C_VEL
LIN {X 0,Y 509.826,Z 129.978,A -85,B 0,C 180,E1 -5633.692,E2 -5633.692} C_VEL
LIN {X 0,Y 509.156,Z 130.063,A -85,B 0,C 180,E1 -5634.352,E2 -5634.352} C_VEL
LIN {X 0,Y 506.347,Z 130.41,A -85,B 0,C 180,E1 -5635.424,E2 -5635.424} C_VEL
LIN {X 0,Y 503.963,Z 130.71,A -85,B 0,C 180,E1 -5636.287,E2 -5636.287} C_VEL
LIN {X 0,Y 502.915,Z 130.836,A -85,B 0,C 180,E1 -5636.954,E2 -5636.954} C_VEL
LIN {X 0,Y 502.816,Z 130.848,A -85,B 0,C 180,E1 -5637.179,E2 -5637.179} C_VEL
LIN {X 0,Y 502.819,Z 130.853,A -85,B 0,C 180,E1 -5640.065,E2 -5640.065} C_VEL
LIN {X 0,Y 502.832,Z 130.85,A -85,B 0,C 180,E1 -5642.533,E2 -5642.533} C_VEL
LIN {X 0,Y 502.843,Z 130.87,A -85,B 0,C 180,E1 -5645.617,E2 -5645.617} C_VEL
LIN {X 0,Y 503.536,Z 135.398,A -85,B 0,C 180,E1 -5646.56,E2 -5646.56} C_VEL
LIN {X 0,Y 503.341,Z 148.945,A -85,B 0,C 180,E1 -5649.238,E2 -5649.238} C_VEL
LIN {X 0,Y 505.481,Z 160.303,A -85,B 0,C 180,E1 -5649.481,E2 -5649.481} C_VEL
LIN {X 0,Y 504.955,Z 256.508,A -85,B 0,C 180,E1 -5650.882,E2 -5650.882} C_VEL
LIN {X 0,Y 504.701,Z 269.824,A -85,B 0,C 180,E1 -5651.247,E2 -5651.247} C_VEL
LIN {X 0,Y 504.477,Z 281.891,A -85,B 0,C 180,E1 -5651.736,E2 -5651.736} C_VEL
LIN {X 0,Y 504.176,Z 293.18,A -85,B 0,C 180,E1 -5652.35,E2 -5652.35} C_VEL
LIN {X 0,Y 503.786,Z 304.893,A -85,B 0,C 180,E1 -5653.173,E2 -5653.173} C_VEL
LIN {X 0,Y 503.448,Z 315.398,A -85,B 0,C 180,E1 -5654.1,E2 -5654.1} C_VEL
LIN {X 0,Y 503.192,Z 323.942,A -85,B 0,C 180,E1 -5655.025,E2 -5655.025} C_VEL
LIN {X 0,Y 502.82,Z 333.143,A -85,B 0,C 180,E1 -5656.254,E2 -5656.254} C_VEL
LIN {X 0,Y 502.576,Z 340.519,A -85,B 0,C 180,E1 -5657.481,E2 -5657.481} C_VEL
LIN {X 0,Y 502.398,Z 346.404,A -85,B 0,C 180,E1 -5658.705,E2 -5658.705} C_VEL
LIN {X 0,Y 502.253,Z 351.02,A -85,B 0,C 180,E1 -5659.926,E2 -5659.926} C_VEL
LIN {X 0,Y 502.175,Z 354.516,A -85,B 0,C 180,E1 -5661.144,E2 -5661.144} C_VEL
LIN {X 0,Y 502.16,Z 356.271,A -85,B 0,C 180,E1 -5661.954,E2 -5661.954} C_VEL
LIN {X 0,Y 502.189,Z 358.525,A -85,B 0,C 180,E1 -5663.571,E2 -5663.571} C_VEL
LIN {X 0,Y 502.155,Z 359.069,A -85,B 0,C 180,E1 -5664.377,E2 -5664.377} C_VEL
LIN {X 0,Y 502.069,Z 359.186,A -85,B 0,C 180,E1 -5665.181,E2 -5665.181} C_VEL
LIN {X 0,Y 502.16,Z 358.905,A -85,B 0,C 180,E1 -5665.987,E2 -5665.987} C_VEL
LIN {X 0,Y 502.168,Z 358.249,A -85,B 0,C 180,E1 -5666.79,E2 -5666.79} C_VEL
LIN {X 0,Y 502.13,Z 357.213,A -85,B 0,C 180,E1 -5667.593,E2 -5667.593} C_VEL
LIN {X 0,Y 502.057,Z 355.74,A -85,B 0,C 180,E1 -5668.395,E2 -5668.395} C_VEL
LIN {X 0,Y 502.185,Z 352.749,A -85,B 0,C 180,E1 -5669.598,E2 -5669.598} C_VEL
LIN {X 0,Y 502.212,Z 348.737,A -85,B 0,C 180,E1 -5670.801,E2 -5670.801} C_VEL
LIN {X 0,Y 502.437,Z 343.567,A -85,B 0,C 180,E1 -5672.003,E2 -5672.003} C_VEL
LIN {X 0,Y 502.544,Z 337.106,A -85,B 0,C 180,E1 -5673.206,E2 -5673.206} C_VEL
LIN {X 0,Y 502.783,Z 330.542,A -85,B 0,C 180,E1 -5674.208,E2 -5674.208} C_VEL
LIN {X 0,Y 503.158,Z 322.625,A -85,B 0,C 180,E1 -5675.208,E2 -5675.208} C_VEL
LIN {X 0,Y 503.525,Z 312.989,A -85,B 0,C 180,E1 -5676.209,E2 -5676.209} C_VEL
LIN {X 0,Y 503.962,Z 302.256,A -85,B 0,C 180,E1 -5677.109,E2 -5677.109} C_VEL
LIN {X 0,Y 504.262,Z 291.787,A -85,B 0,C 180,E1 -5677.809,E2 -5677.809} C_VEL
LIN {X 0,Y 504.533,Z 279.629,A -85,B 0,C 180,E1 -5678.442,E2 -5678.442} C_VEL
LIN {X 0,Y 504.764,Z 266.62,A -85,B 0,C 180,E1 -5678.935,E2 -5678.935} C_VEL
LIN {X 0,Y 504.901,Z 254.517,A -85,B 0,C 180,E1 -5679.236,E2 -5679.236} C_VEL
LIN {X 0,Y 505.499,Z 160.211,A -85,B 0,C 180,E1 -5680.589,E2 -5680.589} C_VEL
LIN {X 0,Y 503.251,Z 148.82,A -85,B 0,C 180,E1 -5680.841,E2 -5680.841} C_VEL
LIN {X 0,Y 503.464,Z 135.2,A -85,B 0,C 180,E1 -5683.521,E2 -5683.521} C_VEL
LIN {X 0,Y 502.911,Z 130.844,A -85,B 0,C 180,E1 -5684.439,E2 -5684.439} C_VEL
LIN {X 0,Y 502.824,Z 130.852,A -85,B 0,C 180,E1 -5687.907,E2 -5687.907} C_VEL
LIN {X 0,Y 502.83,Z 130.851,A -85,B 0,C 180,E1 -5690.535,E2 -5690.535} C_VEL
LIN {X 0,Y 502.788,Z 130.852,A -85,B 0,C 180,E1 -5693.04,E2 -5693.04} C_VEL
LIN {X 0,Y 502.821,Z 130.85,A -85,B 0,C 180,E1 -5695.675,E2 -5695.675} C_VEL
LIN {X 0,Y 502.835,Z 130.849,A -85,B 0,C 180,E1 -5698.372,E2 -5698.372} C_VEL
LIN {X 0,Y 502.791,Z 130.854,A -85,B 0,C 180,E1 -5701.498,E2 -5701.498} C_VEL
LIN {X 0,Y 502.801,Z 130.856,A -85,B 0,C 180,E1 -5703.993,E2 -5703.993} C_VEL
LIN {X 0,Y 502.774,Z 130.856,A -85,B 0,C 180,E1 -5707.177,E2 -5707.177} C_VEL
LIN {X 0,Y 502.783,Z 130.856,A -85,B 0,C 180,E1 -5710.014,E2 -5710.014} C_VEL
LIN {X 0,Y 502.798,Z 130.852,A -85,B 0,C 180,E1 -5712.198,E2 -5712.198} C_VEL
LIN {X 0,Y 502.78,Z 130.859,A -85,B 0,C 180,E1 -5715.469,E2 -5715.469} C_VEL
LIN {X 0,Y 502.812,Z 130.852,A -85,B 0,C 180,E1 -5718.933,E2 -5718.933} C_VEL
LIN {X 0,Y 502.784,Z 130.854,A -85,B 0,C 180,E1 -5722.045,E2 -5722.045} C_VEL
LIN {X 0,Y 502.786,Z 130.857,A -85,B 0,C 180,E1 -5725.033,E2 -5725.033} C_VEL
LIN {X 0,Y 502.772,Z 130.855,A -85,B 0,C 180,E1 -5727.914,E2 -5727.914} C_VEL
LIN {X 0,Y 502.812,Z 130.853,A -85,B 0,C 180,E1 -5730.711,E2 -5730.711} C_VEL
LIN {X 0,Y 502.834,Z 130.849,A -85,B 0,C 180,E1 -5733.443,E2 -5733.443} C_VEL
LIN {X 0,Y 502.774,Z 130.86,A -85,B 0,C 180,E1 -5736.958,E2 -5736.958} C_VEL
LIN {X 0,Y 502.822,Z 130.849,A -85,B 0,C 180,E1 -5739.547,E2 -5739.547} C_VEL
LIN {X 0,Y 502.789,Z 130.856,A -85,B 0,C 180,E1 -5742.09,E2 -5742.09} C_VEL
LIN {X 0,Y 502.813,Z 130.85,A -85,B 0,C 180,E1 -5745.428,E2 -5745.428} C_VEL
LIN {X 0,Y 502.863,Z 130.848,A -85,B 0,C 180,E1 -5748.716,E2 -5748.716} C_VEL
LIN {X 0,Y 502.858,Z 130.849,A -85,B 0,C 180,E1 -5751.966,E2 -5751.966} C_VEL
LIN {X 0,Y 502.883,Z 130.846,A -85,B 0,C 180,E1 -5754.386,E2 -5754.386} C_VEL
LIN {X 0,Y 502.996,Z 130.83,A -85,B 0,C 180,E1 -5757.598,E2 -5757.598} C_VEL
LIN {X 0,Y 502.99,Z 130.832,A -85,B 0,C 180,E1 -5760,E2 -5760} C_VEL
LIN {X 0,Y 502.997,Z 130.83,A -85,B 0,C 180,E1 -5762.402,E2 -5762.402} C_VEL
LIN {X 0,Y 502.89,Z 130.845,A -85,B 0,C 180,E1 -5765.614,E2 -5765.614} C_VEL
LIN {X 0,Y 502.848,Z 130.846,A -85,B 0,C 180,E1 -5768.844,E2 -5768.844} C_VEL
LIN {X 0,Y 502.831,Z 130.85,A -85,B 0,C 180,E1 -5772.102,E2 -5772.102} C_VEL
LIN {X 0,Y 502.836,Z 130.852,A -85,B 0,C 180,E1 -5775.4,E2 -5775.4} C_VEL
LIN {X 0,Y 502.809,Z 130.852,A -85,B 0,C 180,E1 -5778.753,E2 -5778.753} C_VEL
LIN {X 0,Y 502.769,Z 130.859,A -85,B 0,C 180,E1 -5781.312,E2 -5781.312} C_VEL
LIN {X 0,Y 502.755,Z 130.858,A -85,B 0,C 180,E1 -5783.916,E2 -5783.916} C_VEL
LIN {X 0,Y 502.825,Z 130.85,A -85,B 0,C 180,E1 -5786.568,E2 -5786.568} C_VEL
LIN {X 0,Y 502.811,Z 130.853,A -85,B 0,C 180,E1 -5789.289,E2 -5789.289} C_VEL
LIN {X 0,Y 502.772,Z 130.855,A -85,B 0,C 180,E1 -5792.086,E2 -5792.086} C_VEL
LIN {X 0,Y 502.786,Z 130.857,A -85,B 0,C 180,E1 -5794.967,E2 -5794.967} C_VEL
LIN {X 0,Y 502.784,Z 130.853,A -85,B 0,C 180,E1 -5797.955,E2 -5797.955} C_VEL
LIN {X 0,Y 502.811,Z 130.852,A -85,B 0,C 180,E1 -5801.067,E2 -5801.067} C_VEL
LIN {X 0,Y 502.779,Z 130.859,A -85,B 0,C 180,E1 -5804.531,E2 -5804.531} C_VEL
LIN {X 0,Y 502.788,Z 130.854,A -85,B 0,C 180,E1 -5807.862,E2 -5807.862} C_VEL
LIN {X 0,Y 502.796,Z 130.852,A -85,B 0,C 180,E1 -5811.025,E2 -5811.025} C_VEL
LIN {X 0,Y 502.77,Z 130.862,A -85,B 0,C 180,E1 -5814.17,E2 -5814.17} C_VEL
LIN {X 0,Y 502.829,Z 130.847,A -85,B 0,C 180,E1 -5816.994,E2 -5816.994} C_VEL
LIN {X 0,Y 502.812,Z 130.856,A -85,B 0,C 180,E1 -5820.066,E2 -5820.066} C_VEL
LIN {X 0,Y 502.83,Z 130.848,A -85,B 0,C 180,E1 -5822.534,E2 -5822.534} C_VEL
LIN {X 0,Y 502.862,Z 130.92,A -85,B 0,C 180,E1 -5824.604,E2 -5824.604} C_VEL
LIN {X 0,Y 504.552,Z 140.267,A -85,B 0,C 180,E1 -5826.176,E2 -5826.176} C_VEL
LIN {X 0,Y 504.071,Z 158.096,A -85,B 0,C 180,E1 -5828.981,E2 -5828.981} C_VEL
LIN {X 0,Y 503.568,Z 178.304,A -85,B 0,C 180,E1 -5832.12,E2 -5832.12} C_VEL
LIN {X 0,Y 503.208,Z 191.887,A -85,B 0,C 180,E1 -5834.198,E2 -5834.198} C_VEL
LIN {X 0,Y 505.322,Z 207.695,A -85,B 0,C 180,E1 -5834.49,E2 -5834.49} C_VEL
LIN {X 0,Y 504.825,Z 300.233,A -85,B 0,C 180,E1 -5835.823,E2 -5835.823} C_VEL
LIN {X 0,Y 504.584,Z 312.827,A -85,B 0,C 180,E1 -5836.15,E2 -5836.15} C_VEL
LIN {X 0,Y 504.215,Z 325.808,A -85,B 0,C 180,E1 -5836.653,E2 -5836.653} C_VEL
LIN {X 0,Y 503.843,Z 338.025,A -85,B 0,C 180,E1 -5837.303,E2 -5837.303} C_VEL
LIN {X 0,Y 503.464,Z 349.764,A -85,B 0,C 180,E1 -5838.119,E2 -5838.119} C_VEL
LIN {X 0,Y 503.187,Z 360.244,A -85,B 0,C 180,E1 -5839.031,E2 -5839.031} C_VEL
LIN {X 0,Y 502.818,Z 368.808,A -85,B 0,C 180,E1 -5839.939,E2 -5839.939} C_VEL
LIN {X 0,Y 502.593,Z 376.714,A -85,B 0,C 180,E1 -5840.95,E2 -5840.95} C_VEL
LIN {X 0,Y 502.363,Z 384.436,A -85,B 0,C 180,E1 -5842.161,E2 -5842.161} C_VEL
LIN {X 0,Y 502.214,Z 391.558,A -85,B 0,C 180,E1 -5843.573,E2 -5843.573} C_VEL
LIN {X 0,Y 502.171,Z 396.298,A -85,B 0,C 180,E1 -5844.781,E2 -5844.781} C_VEL
LIN {X 0,Y 502.139,Z 399.919,A -85,B 0,C 180,E1 -5845.988,E2 -5845.988} C_VEL
LIN {X 0,Y 502.137,Z 401.787,A -85,B 0,C 180,E1 -5846.791,E2 -5846.791} C_VEL
LIN {X 0,Y 502.124,Z 403.187,A -85,B 0,C 180,E1 -5847.594,E2 -5847.594} C_VEL
LIN {X 0,Y 502.001,Z 404.789,A -85,B 0,C 180,E1 -5849.199,E2 -5849.199} C_VEL
LIN {X 0,Y 501.997,Z 405.004,A -85,B 0,C 180,E1 -5850.001,E2 -5850.001} C_VEL
LIN {X 0,Y 502.037,Z 404.175,A -85,B 0,C 180,E1 -5851.605,E2 -5851.605} C_VEL
LIN {X 0,Y 502.125,Z 403.178,A -85,B 0,C 180,E1 -5852.407,E2 -5852.407} C_VEL
LIN {X 0,Y 502.137,Z 401.775,A -85,B 0,C 180,E1 -5853.21,E2 -5853.21} C_VEL
LIN {X 0,Y 502.101,Z 398.822,A -85,B 0,C 180,E1 -5854.416,E2 -5854.416} C_VEL
LIN {X 0,Y 502.189,Z 394.832,A -85,B 0,C 180,E1 -5855.623,E2 -5855.623} C_VEL
LIN {X 0,Y 502.282,Z 388.796,A -85,B 0,C 180,E1 -5857.013,E2 -5857.013} C_VEL
LIN {X 0,Y 502.446,Z 381.991,A -85,B 0,C 180,E1 -5858.244,E2 -5858.244} C_VEL
LIN {X 0,Y 502.684,Z 373.677,A -85,B 0,C 180,E1 -5859.456,E2 -5859.456} C_VEL
LIN {X 0,Y 502.95,Z 365.162,A -85,B 0,C 180,E1 -5860.467,E2 -5860.467} C_VEL
LIN {X 0,Y 503.308,Z 354.647,A -85,B 0,C 180,E1 -5861.478,E2 -5861.478} C_VEL
LIN {X 0,Y 503.661,Z 343.04,A -85,B 0,C 180,E1 -5862.373,E2 -5862.373} C_VEL
LIN {X 0,Y 504.038,Z 330.946,A -85,B 0,C 180,E1 -5863.096,E2 -5863.096} C_VEL
LIN {X 0,Y 504.393,Z 318.604,A -85,B 0,C 180,E1 -5863.651,E2 -5863.651} C_VEL
LIN {X 0,Y 504.706,Z 305.958,A -85,B 0,C 180,E1 -5864.053,E2 -5864.053} C_VEL
LIN {X 0,Y 504.904,Z 292.817,A -85,B 0,C 180,E1 -5864.305,E2 -5864.305} C_VEL
LIN {X 0,Y 505.193,Z 205.26,A -85,B 0,C 180,E1 -5865.56,E2 -5865.56} C_VEL
LIN {X 0,Y 503.225,Z 191.577,A -85,B 0,C 180,E1 -5865.844,E2 -5865.844} C_VEL
LIN {X 0,Y 503.739,Z 171.692,A -85,B 0,C 180,E1 -5868.928,E2 -5868.928} C_VEL
LIN {X 0,Y 504.26,Z 152.871,A -85,B 0,C 180,E1 -5871.89,E2 -5871.89} C_VEL
LIN {X 0,Y 504.671,Z 140.771,A -85,B 0,C 180,E1 -5873.82,E2 -5873.82} C_VEL
LIN {X 0,Y 502.837,Z 130.85,A -85,B 0,C 180,E1 -5875.566,E2 -5875.566} C_VEL
LIN {X 0,Y 502.8,Z 130.858,A -85,B 0,C 180,E1 -5878.376,E2 -5878.376} C_VEL
LIN {X 0,Y 502.797,Z 130.855,A -85,B 0,C 180,E1 -5881.144,E2 -5881.144} C_VEL
LIN {X 0,Y 502.806,Z 130.855,A -85,B 0,C 180,E1 -5883.994,E2 -5883.994} C_VEL
LIN {X 0,Y 502.767,Z 130.855,A -85,B 0,C 180,E1 -5887.176,E2 -5887.176} C_VEL
LIN {X 0,Y 502.789,Z 130.854,A -85,B 0,C 180,E1 -5890.015,E2 -5890.015} C_VEL
LIN {X 0,Y 502.805,Z 130.85,A -85,B 0,C 180,E1 -5892.199,E2 -5892.199} C_VEL
LIN {X 0,Y 502.787,Z 130.859,A -85,B 0,C 180,E1 -5895.47,E2 -5895.47} C_VEL
LIN {X 0,Y 502.796,Z 130.853,A -85,B 0,C 180,E1 -5897.861,E2 -5897.861} C_VEL
LIN {X 0,Y 502.794,Z 130.857,A -85,B 0,C 180,E1 -5901.023,E2 -5901.023} C_VEL
LIN {X 0,Y 502.774,Z 130.854,A -85,B 0,C 180,E1 -5904.169,E2 -5904.169} C_VEL
LIN {X 0,Y 502.831,Z 130.854,A -85,B 0,C 180,E1 -5906.994,E2 -5906.994} C_VEL
LIN {X 0,Y 502.809,Z 130.849,A -85,B 0,C 180,E1 -5910.066,E2 -5910.066} C_VEL
LIN {X 0,Y 502.774,Z 130.854,A -85,B 0,C 180,E1 -5913.46,E2 -5913.46} C_VEL
LIN {X 0,Y 502.764,Z 130.855,A -85,B 0,C 180,E1 -5916.085,E2 -5916.085} C_VEL
LIN {X 0,Y 502.83,Z 130.844,A -85,B 0,C 180,E1 -5919.464,E2 -5919.464} C_VEL
LIN {X 0,Y 502.784,Z 130.853,A -85,B 0,C 180,E1 -5922.09,E2 -5922.09} C_VEL
LIN {X 0,Y 502.821,Z 130.844,A -85,B 0,C 180,E1 -5925.428,E2 -5925.428} C_VEL
LIN {X 0,Y 502.833,Z 130.848,A -85,B 0,C 180,E1 -5928.716,E2 -5928.716} C_VEL
LIN {X 0,Y 502.844,Z 130.846,A -85,B 0,C 180,E1 -5931.966,E2 -5931.966} C_VEL
LIN {X 0,Y 502.888,Z 130.843,A -85,B 0,C 180,E1 -5934.386,E2 -5934.386} C_VEL
LIN {X 0,Y 503.006,Z 130.823,A -85,B 0,C 180,E1 -5937.598,E2 -5937.598} C_VEL
LIN {X 0,Y 503.001,Z 130.832,A -85,B 0,C 180,E1 -5940,E2 -5940} C_VEL
LIN {X 0,Y 503.007,Z 130.821,A -85,B 0,C 180,E1 -5942.402,E2 -5942.402} C_VEL
LIN {X 0,Y 502.891,Z 130.845,A -85,B 0,C 180,E1 -5945.614,E2 -5945.614} C_VEL
LIN {X 0,Y 502.855,Z 130.841,A -85,B 0,C 180,E1 -5948.034,E2 -5948.034} C_VEL
LIN {X 0,Y 502.875,Z 130.845,A -85,B 0,C 180,E1 -5951.283,E2 -5951.283} C_VEL
LIN {X 0,Y 502.825,Z 130.843,A -85,B 0,C 180,E1 -5954.572,E2 -5954.572} C_VEL
LIN {X 0,Y 502.816,Z 130.848,A -85,B 0,C 180,E1 -5957.909,E2 -5957.909} C_VEL
LIN {X 0,Y 502.83,Z 130.845,A -85,B 0,C 180,E1 -5960.536,E2 -5960.536} C_VEL
LIN {X 0,Y 502.786,Z 130.859,A -85,B 0,C 180,E1 -5963.041,E2 -5963.041} C_VEL
LIN {X 0,Y 502.836,Z 130.848,A -85,B 0,C 180,E1 -5966.568,E2 -5966.568} C_VEL
LIN {X 0,Y 502.815,Z 130.847,A -85,B 0,C 180,E1 -5969.935,E2 -5969.935} C_VEL
LIN {X 0,Y 502.831,Z 130.85,A -85,B 0,C 180,E1 -5973.032,E2 -5973.032} C_VEL
LIN {X 0,Y 502.775,Z 130.853,A -85,B 0,C 180,E1 -5975.951,E2 -5975.951} C_VEL
LIN {X 0,Y 502.798,Z 130.851,A -85,B 0,C 180,E1 -5978.977,E2 -5978.977} C_VEL
LIN {X 0,Y 502.822,Z 130.842,A -85,B 0,C 180,E1 -5981.066,E2 -5981.066} C_VEL
LIN {X 0,Y 502.789,Z 130.857,A -85,B 0,C 180,E1 -5984.53,E2 -5984.53} C_VEL
LIN {X 0,Y 502.798,Z 130.853,A -85,B 0,C 180,E1 -5987.861,E2 -5987.861} C_VEL
LIN {X 0,Y 502.805,Z 130.85,A -85,B 0,C 180,E1 -5991.024,E2 -5991.024} C_VEL
LIN {X 0,Y 502.779,Z 130.86,A -85,B 0,C 180,E1 -5994.169,E2 -5994.169} C_VEL
LIN {X 0,Y 502.816,Z 130.848,A -85,B 0,C 180,E1 -5997.179,E2 -5997.179} C_VEL
LIN {X 0,Y 502.112,Z 130.943,A -85,B 0,C 180,E1 -5997.848,E2 -5997.848} C_VEL
LIN {X 0,Y 499.248,Z 131.295,A -85,B 0,C 180,E1 -5998.934,E2 -5998.934} C_VEL
LIN {X 0,Y 496.854,Z 131.598,A -85,B 0,C 180,E1 -5999.808,E2 -5999.808} C_VEL
LIN {X 0,Y 495.835,Z 131.721,A -85,B 0,C 180,E1 -6000.484,E2 -6000.484} C_VEL
LIN {X 0,Y 495.756,Z 131.73,A -85,B 0,C 180,E1 -6000.713,E2 -6000.713} C_VEL
LIN {X 0,Y 495.828,Z 131.724,A -85,B 0,C 180,E1 -6003.251,E2 -6003.251} C_VEL
LIN {X 0,Y 495.826,Z 131.759,A -85,B 0,C 180,E1 -6005.461,E2 -6005.461} C_VEL
LIN {X 0,Y 496.574,Z 137.455,A -85,B 0,C 180,E1 -6006.654,E2 -6006.654} C_VEL
LIN {X 0,Y 496.409,Z 149.177,A -85,B 0,C 180,E1 -6008.988,E2 -6008.988} C_VEL
LIN {X 0,Y 498.627,Z 160.33,A -85,B 0,C 180,E1 -6009.245,E2 -6009.245} C_VEL
LIN {X 0,Y 498.13,Z 256.364,A -85,B 0,C 180,E1 -6010.663,E2 -6010.663} C_VEL
LIN {X 0,Y 497.845,Z 269.671,A -85,B 0,C 180,E1 -6011.026,E2 -6011.026} C_VEL
LIN {X 0,Y 497.621,Z 281.817,A -85,B 0,C 180,E1 -6011.521,E2 -6011.521} C_VEL
LIN {X 0,Y 497.259,Z 294.136,A -85,B 0,C 180,E1 -6012.203,E2 -6012.203} C_VEL
LIN {X 0,Y 496.847,Z 305.726,A -85,B 0,C 180,E1 -6013.037,E2 -6013.037} C_VEL
LIN {X 0,Y 496.49,Z 316.131,A -85,B 0,C 180,E1 -6013.976,E2 -6013.976} C_VEL
LIN {X 0,Y 496.18,Z 325.427,A -85,B 0,C 180,E1 -6015.02,E2 -6015.02} C_VEL
LIN {X 0,Y 495.784,Z 334.399,A -85,B 0,C 180,E1 -6016.264,E2 -6016.264} C_VEL
LIN {X 0,Y 495.526,Z 341.599,A -85,B 0,C 180,E1 -6017.508,E2 -6017.508} C_VEL
LIN {X 0,Y 495.369,Z 346.433,A -85,B 0,C 180,E1 -6018.543,E2 -6018.543} C_VEL
LIN {X 0,Y 495.204,Z 351.11,A -85,B 0,C 180,E1 -6019.781,E2 -6019.781} C_VEL
LIN {X 0,Y 495.105,Z 354.664,A -85,B 0,C 180,E1 -6021.016,E2 -6021.016} C_VEL
LIN {X 0,Y 495.096,Z 356.475,A -85,B 0,C 180,E1 -6021.839,E2 -6021.839} C_VEL
LIN {X 0,Y 495.107,Z 358.782,A -85,B 0,C 180,E1 -6023.479,E2 -6023.479} C_VEL
LIN {X 0,Y 495.074,Z 359.355,A -85,B 0,C 180,E1 -6024.296,E2 -6024.296} C_VEL
LIN {X 0,Y 494.992,Z 359.523,A -85,B 0,C 180,E1 -6025.112,E2 -6025.112} C_VEL
LIN {X 0,Y 495.058,Z 359.269,A -85,B 0,C 180,E1 -6025.929,E2 -6025.929} C_VEL
LIN {X 0,Y 495.086,Z 358.638,A -85,B 0,C 180,E1 -6026.744,E2 -6026.744} C_VEL
LIN {X 0,Y 495.064,Z 357.629,A -85,B 0,C 180,E1 -6027.558,E2 -6027.558} C_VEL
LIN {X 0,Y 494.983,Z 356.209,A -85,B 0,C 180,E1 -6028.372,E2 -6028.372} C_VEL
LIN {X 0,Y 495.112,Z 353.271,A -85,B 0,C 180,E1 -6029.593,E2 -6029.593} C_VEL
LIN {X 0,Y 495.137,Z 349.316,A -85,B 0,C 180,E1 -6030.813,E2 -6030.813} C_VEL
LIN {X 0,Y 495.369,Z 344.215,A -85,B 0,C 180,E1 -6032.032,E2 -6032.032} C_VEL
LIN {X 0,Y 495.492,Z 337.819,A -85,B 0,C 180,E1 -6033.252,E2 -6033.252} C_VEL
LIN {X 0,Y 495.744,Z 331.33,A -85,B 0,C 180,E1 -6034.268,E2 -6034.268} C_VEL
LIN {X 0,Y 496.138,Z 323.5,A -85,B 0,C 180,E1 -6035.282,E2 -6035.282} C_VEL
LIN {X 0,Y 496.528,Z 313.969,A -85,B 0,C 180,E1 -6036.297,E2 -6036.297} C_VEL
LIN {X 0,Y 496.969,Z 303.384,A -85,B 0,C 180,E1 -6037.209,E2 -6037.209} C_VEL
LIN {X 0,Y 497.309,Z 293.141,A -85,B 0,C 180,E1 -6037.919,E2 -6037.919} C_VEL
LIN {X 0,Y 497.587,Z 281.59,A -85,B 0,C 180,E1 -6038.547,E2 -6038.547} C_VEL
LIN {X 0,Y 497.835,Z 268.761,A -85,B 0,C 180,E1 -6039.061,E2 -6039.061} C_VEL
LIN {X 0,Y 498.021,Z 255.405,A -85,B 0,C 180,E1 -6039.416,E2 -6039.416} C_VEL
LIN {X 0,Y 498.634,Z 160.847,A -85,B 0,C 180,E1 -6040.793,E2 -6040.793} C_VEL
LIN {X 0,Y 496.273,Z 149.145,A -85,B 0,C 180,E1 -6041.047,E2 -6041.047} C_VEL
LIN {X 0,Y 496.427,Z 135.677,A -85,B 0,C 180,E1 -6043.716,E2 -6043.716} C_VEL
LIN {X 0,Y 495.858,Z 131.723,A -85,B 0,C 180,E1 -6044.57,E2 -6044.57} C_VEL
LIN {X 0,Y 495.782,Z 131.731,A -85,B 0,C 180,E1 -6048.17,E2 -6048.17} C_VEL
LIN {X 0,Y 495.775,Z 131.727,A -85,B 0,C 180,E1 -6050.755,E2 -6050.755} C_VEL
LIN {X 0,Y 495.743,Z 131.73,A -85,B 0,C 180,E1 -6053.386,E2 -6053.386} C_VEL
LIN {X 0,Y 495.822,Z 131.72,A -85,B 0,C 180,E1 -6056.748,E2 -6056.748} C_VEL
LIN {X 0,Y 495.764,Z 131.731,A -85,B 0,C 180,E1 -6059.745,E2 -6059.745} C_VEL
LIN {X 0,Y 495.765,Z 131.728,A -85,B 0,C 180,E1 -6062.593,E2 -6062.593} C_VEL
LIN {X 0,Y 495.744,Z 131.733,A -85,B 0,C 180,E1 -6065.536,E2 -6065.536} C_VEL
LIN {X 0,Y 495.759,Z 131.728,A -85,B 0,C 180,E1 -6068.767,E2 -6068.767} C_VEL
LIN {X 0,Y 495.751,Z 131.735,A -85,B 0,C 180,E1 -6071.78,E2 -6071.78} C_VEL
LIN {X 0,Y 495.731,Z 131.734,A -85,B 0,C 180,E1 -6075.14,E2 -6075.14} C_VEL
LIN {X 0,Y 495.749,Z 131.73,A -85,B 0,C 180,E1 -6078.218,E2 -6078.218} C_VEL
LIN {X 0,Y 495.742,Z 131.737,A -85,B 0,C 180,E1 -6081.407,E2 -6081.407} C_VEL
LIN {X 0,Y 495.738,Z 131.732,A -85,B 0,C 180,E1 -6084.461,E2 -6084.461} C_VEL
LIN {X 0,Y 495.757,Z 131.733,A -85,B 0,C 180,E1 -6087.405,E2 -6087.405} C_VEL
LIN {X 0,Y 495.755,Z 131.73,A -85,B 0,C 180,E1 -6090.253,E2 -6090.253} C_VEL
LIN {X 0,Y 495.795,Z 131.728,A -85,B 0,C 180,E1 -6093.254,E2 -6093.254} C_VEL
LIN {X 0,Y 495.727,Z 131.736,A -85,B 0,C 180,E1 -6096.611,E2 -6096.611} C_VEL
LIN {X 0,Y 495.767,Z 131.729,A -85,B 0,C 180,E1 -6099.324,E2 -6099.324} C_VEL
LIN {X 0,Y 495.767,Z 131.729,A -85,B 0,C 180,E1 -6101.828,E2 -6101.828} C_VEL
LIN {X 0,Y 495.764,Z 131.729,A -85,B 0,C 180,E1 -6105.216,E2 -6105.216} C_VEL
LIN {X 0,Y 495.838,Z 131.723,A -85,B 0,C 180,E1 -6108.554,E2 -6108.554} C_VEL
LIN {X 0,Y 495.817,Z 131.725,A -85,B 0,C 180,E1 -6111.851,E2 -6111.851} C_VEL
LIN {X 0,Y 495.807,Z 131.723,A -85,B 0,C 180,E1 -6115.121,E2 -6115.121} C_VEL
LIN {X 0,Y 495.963,Z 131.706,A -85,B 0,C 180,E1 -6117.563,E2 -6117.563} C_VEL
LIN {X 0,Y 495.959,Z 131.707,A -85,B 0,C 180,E1 -6120,E2 -6120} C_VEL
LIN {X 0,Y 495.964,Z 131.706,A -85,B 0,C 180,E1 -6122.436,E2 -6122.436} C_VEL
LIN {X 0,Y 495.848,Z 131.722,A -85,B 0,C 180,E1 -6125.694,E2 -6125.694} C_VEL
LIN {X 0,Y 495.818,Z 131.723,A -85,B 0,C 180,E1 -6128.97,E2 -6128.97} C_VEL
LIN {X 0,Y 495.816,Z 131.725,A -85,B 0,C 180,E1 -6132.035,E2 -6132.035} C_VEL
LIN {X 0,Y 495.811,Z 131.726,A -85,B 0,C 180,E1 -6135.451,E2 -6135.451} C_VEL
LIN {X 0,Y 495.765,Z 131.732,A -85,B 0,C 180,E1 -6139.029,E2 -6139.029} C_VEL
LIN {X 0,Y 495.729,Z 131.735,A -85,B 0,C 180,E1 -6141.63,E2 -6141.63} C_VEL
LIN {X 0,Y 495.701,Z 131.736,A -85,B 0,C 180,E1 -6144.278,E2 -6144.278} C_VEL
LIN {X 0,Y 495.772,Z 131.732,A -85,B 0,C 180,E1 -6146.977,E2 -6146.977} C_VEL
LIN {X 0,Y 495.755,Z 131.73,A -85,B 0,C 180,E1 -6149.747,E2 -6149.747} C_VEL
LIN {X 0,Y 495.756,Z 131.733,A -85,B 0,C 180,E1 -6152.595,E2 -6152.595} C_VEL
LIN {X 0,Y 495.737,Z 131.732,A -85,B 0,C 180,E1 -6155.539,E2 -6155.539} C_VEL
LIN {X 0,Y 495.754,Z 131.733,A -85,B 0,C 180,E1 -6158.769,E2 -6158.769} C_VEL
LIN {X 0,Y 495.748,Z 131.73,A -85,B 0,C 180,E1 -6161.782,E2 -6161.782} C_VEL
LIN {X 0,Y 495.73,Z 131.733,A -85,B 0,C 180,E1 -6165.142,E2 -6165.142} C_VEL
LIN {X 0,Y 495.749,Z 131.735,A -85,B 0,C 180,E1 -6168.22,E2 -6168.22} C_VEL
LIN {X 0,Y 495.745,Z 131.729,A -85,B 0,C 180,E1 -6171.41,E2 -6171.41} C_VEL
LIN {X 0,Y 495.743,Z 131.733,A -85,B 0,C 180,E1 -6174.463,E2 -6174.463} C_VEL
LIN {X 0,Y 495.764,Z 131.727,A -85,B 0,C 180,E1 -6177.407,E2 -6177.407} C_VEL
LIN {X 0,Y 495.763,Z 131.734,A -85,B 0,C 180,E1 -6180.255,E2 -6180.255} C_VEL
LIN {X 0,Y 495.821,Z 131.721,A -85,B 0,C 180,E1 -6183.252,E2 -6183.252} C_VEL
LIN {X 0,Y 495.835,Z 131.836,A -85,B 0,C 180,E1 -6184.443,E2 -6184.443} C_VEL
LIN {X 0,Y 497.575,Z 141.198,A -85,B 0,C 180,E1 -6186.043,E2 -6186.043} C_VEL
LIN {X 0,Y 497.165,Z 156.192,A -85,B 0,C 180,E1 -6188.437,E2 -6188.437} C_VEL
LIN {X 0,Y 496.59,Z 176.283,A -85,B 0,C 180,E1 -6191.605,E2 -6191.605} C_VEL
LIN {X 0,Y 496.174,Z 191.467,A -85,B 0,C 180,E1 -6193.976,E2 -6193.976} C_VEL
LIN {X 0,Y 498.459,Z 208.014,A -85,B 0,C 180,E1 -6194.289,E2 -6194.289} C_VEL
LIN {X 0,Y 497.9,Z 300.722,A -85,B 0,C 180,E1 -6195.648,E2 -6195.648} C_VEL
LIN {X 0,Y 497.64,Z 313.817,A -85,B 0,C 180,E1 -6196.005,E2 -6196.005} C_VEL
LIN {X 0,Y 497.267,Z 326.465,A -85,B 0,C 180,E1 -6196.516,E2 -6196.516} C_VEL
LIN {X 0,Y 496.884,Z 337.897,A -85,B 0,C 180,E1 -6197.141,E2 -6197.141} C_VEL
LIN {X 0,Y 496.466,Z 349.374,A -85,B 0,C 180,E1 -6197.949,E2 -6197.949} C_VEL
LIN {X 0,Y 496.153,Z 359.875,A -85,B 0,C 180,E1 -6198.873,E2 -6198.873} C_VEL
LIN {X 0,Y 495.8,Z 368.453,A -85,B 0,C 180,E1 -6199.795,E2 -6199.795} C_VEL
LIN {X 0,Y 495.526,Z 376.371,A -85,B 0,C 180,E1 -6200.82,E2 -6200.82} C_VEL
LIN {X 0,Y 495.31,Z 384.105,A -85,B 0,C 180,E1 -6202.049,E2 -6202.049} C_VEL
LIN {X 0,Y 495.134,Z 391.23,A -85,B 0,C 180,E1 -6203.481,E2 -6203.481} C_VEL
LIN {X 0,Y 495.101,Z 395.973,A -85,B 0,C 180,E1 -6204.707,E2 -6204.707} C_VEL
LIN {X 0,Y 495.034,Z 399.594,A -85,B 0,C 180,E1 -6205.93,E2 -6205.93} C_VEL
LIN {X 0,Y 495.056,Z 401.464,A -85,B 0,C 180,E1 -6206.745,E2 -6206.745} C_VEL
LIN {X 0,Y 495.028,Z 402.863,A -85,B 0,C 180,E1 -6207.56,E2 -6207.56} C_VEL
LIN {X 0,Y 494.92,Z 404.466,A -85,B 0,C 180,E1 -6209.187,E2 -6209.187} C_VEL
LIN {X 0,Y 494.914,Z 404.681,A -85,B 0,C 180,E1 -6210.001,E2 -6210.001} C_VEL
LIN {X 0,Y 494.964,Z 403.852,A -85,B 0,C 180,E1 -6211.628,E2 -6211.628} C_VEL
LIN {X 0,Y 495.029,Z 402.854,A -85,B 0,C 180,E1 -6212.442,E2 -6212.442} C_VEL
LIN {X 0,Y 495.057,Z 401.451,A -85,B 0,C 180,E1 -6213.256,E2 -6213.256} C_VEL
LIN {X 0,Y 495.006,Z 398.498,A -85,B 0,C 180,E1 -6214.479,E2 -6214.479} C_VEL
LIN {X 0,Y 495.101,Z 394.508,A -85,B 0,C 180,E1 -6215.703,E2 -6215.703} C_VEL
LIN {X 0,Y 495.236,Z 388.374,A -85,B 0,C 180,E1 -6217.134,E2 -6217.134} C_VEL
LIN {X 0,Y 495.4,Z 381.677,A -85,B 0,C 180,E1 -6218.362,E2 -6218.362} C_VEL
LIN {X 0,Y 495.645,Z 373.374,A -85,B 0,C 180,E1 -6219.591,E2 -6219.591} C_VEL
LIN {X 0,Y 495.954,Z 364.873,A -85,B 0,C 180,E1 -6220.616,E2 -6220.616} C_VEL
LIN {X 0,Y 496.31,Z 354.382,A -85,B 0,C 180,E1 -6221.642,E2 -6221.642} C_VEL
LIN {X 0,Y 496.702,Z 343.029,A -85,B 0,C 180,E1 -6222.533,E2 -6222.533} C_VEL
LIN {X 0,Y 497.132,Z 330.758,A -85,B 0,C 180,E1 -6223.282,E2 -6223.282} C_VEL
LIN {X 0,Y 497.484,Z 318.471,A -85,B 0,C 180,E1 -6223.844,E2 -6223.844} C_VEL
LIN {X 0,Y 497.856,Z 304.97,A -85,B 0,C 180,E1 -6224.277,E2 -6224.277} C_VEL
LIN {X 0,Y 498.068,Z 291.299,A -85,B 0,C 180,E1 -6224.531,E2 -6224.531} C_VEL
LIN {X 0,Y 498.487,Z 207.111,A -85,B 0,C 180,E1 -6225.753,E2 -6225.753} C_VEL
LIN {X 0,Y 496.213,Z 191.309,A -85,B 0,C 180,E1 -6226.075,E2 -6226.075} C_VEL
LIN {X 0,Y 496.753,Z 172.799,A -85,B 0,C 180,E1 -6228.99,E2 -6228.99} C_VEL
LIN {X 0,Y 497.332,Z 155.345,A -85,B 0,C 180,E1 -6231.775,E2 -6231.775} C_VEL
LIN {X 0,Y 497.743,Z 141.913,A -85,B 0,C 180,E1 -6233.95,E2 -6233.95} C_VEL
LIN {X 0,Y 495.8,Z 131.727,A -85,B 0,C 180,E1 -6235.757,E2 -6235.757} C_VEL
LIN {X 0,Y 495.747,Z 131.733,A -85,B 0,C 180,E1 -6238.817,E2 -6238.817} C_VEL
LIN {X 0,Y 495.758,Z 131.736,A -85,B 0,C 180,E1 -6241.725,E2 -6241.725} C_VEL
LIN {X 0,Y 495.77,Z 131.726,A -85,B 0,C 180,E1 -6244.694,E2 -6244.694} C_VEL
LIN {X 0,Y 495.724,Z 131.736,A -85,B 0,C 180,E1 -6247.562,E2 -6247.562} C_VEL
LIN {X 0,Y 495.76,Z 131.729,A -85,B 0,C 180,E1 -6250.047,E2 -6250.047} C_VEL
LIN {X 0,Y 495.719,Z 131.732,A -85,B 0,C 180,E1 -6252.884,E2 -6252.884} C_VEL
LIN {X 0,Y 495.725,Z 131.733,A -85,B 0,C 180,E1 -6255.998,E2 -6255.998} C_VEL
LIN {X 0,Y 495.723,Z 131.733,A -85,B 0,C 180,E1 -6258.712,E2 -6258.712} C_VEL
LIN {X 0,Y 495.746,Z 131.735,A -85,B 0,C 180,E1 -6261.408,E2 -6261.408} C_VEL
LIN {X 0,Y 495.746,Z 131.73,A -85,B 0,C 180,E1 -6264.462,E2 -6264.462} C_VEL
LIN {X 0,Y 495.765,Z 131.73,A -85,B 0,C 180,E1 -6267.405,E2 -6267.405} C_VEL
LIN {X 0,Y 495.756,Z 131.728,A -85,B 0,C 180,E1 -6270.253,E2 -6270.253} C_VEL
LIN {X 0,Y 495.739,Z 131.732,A -85,B 0,C 180,E1 -6273.27,E2 -6273.27} C_VEL
LIN {X 0,Y 495.737,Z 131.736,A -85,B 0,C 180,E1 -6276.612,E2 -6276.612} C_VEL
LIN {X 0,Y 495.779,Z 131.723,A -85,B 0,C 180,E1 -6279.324,E2 -6279.324} C_VEL
LIN {X 0,Y 495.76,Z 131.726,A -85,B 0,C 180,E1 -6281.828,E2 -6281.828} C_VEL
LIN {X 0,Y 495.773,Z 131.722,A -85,B 0,C 180,E1 -6285.217,E2 -6285.217} C_VEL
LIN {X 0,Y 495.812,Z 131.725,A -85,B 0,C 180,E1 -6288.554,E2 -6288.554} C_VEL
LIN {X 0,Y 495.808,Z 131.72,A -85,B 0,C 180,E1 -6291.851,E2 -6291.851} C_VEL
LIN {X 0,Y 495.847,Z 131.721,A -85,B 0,C 180,E1 -6294.306,E2 -6294.306} C_VEL
LIN {X 0,Y 495.972,Z 131.699,A -85,B 0,C 180,E1 -6297.564,E2 -6297.564} C_VEL
LIN {X 0,Y 495.97,Z 131.707,A -85,B 0,C 180,E1 -6300,E2 -6300} C_VEL
LIN {X 0,Y 495.974,Z 131.697,A -85,B 0,C 180,E1 -6302.436,E2 -6302.436} C_VEL
LIN {X 0,Y 495.85,Z 131.723,A -85,B 0,C 180,E1 -6305.694,E2 -6305.694} C_VEL
LIN {X 0,Y 495.819,Z 131.717,A -85,B 0,C 180,E1 -6308.149,E2 -6308.149} C_VEL
LIN {X 0,Y 495.85,Z 131.723,A -85,B 0,C 180,E1 -6311.445,E2 -6311.445} C_VEL
LIN {X 0,Y 495.776,Z 131.722,A -85,B 0,C 180,E1 -6314.783,E2 -6314.783} C_VEL
LIN {X 0,Y 495.779,Z 131.723,A -85,B 0,C 180,E1 -6318.172,E2 -6318.172} C_VEL
LIN {X 0,Y 495.775,Z 131.726,A -85,B 0,C 180,E1 -6320.757,E2 -6320.757} C_VEL
LIN {X 0,Y 495.739,Z 131.731,A -85,B 0,C 180,E1 -6323.388,E2 -6323.388} C_VEL
LIN {X 0,Y 495.775,Z 131.73,A -85,B 0,C 180,E1 -6326.738,E2 -6326.738} C_VEL
LIN {X 0,Y 495.763,Z 131.726,A -85,B 0,C 180,E1 -6329.747,E2 -6329.747} C_VEL
LIN {X 0,Y 495.767,Z 131.731,A -85,B 0,C 180,E1 -6332.595,E2 -6332.595} C_VEL
LIN {X 0,Y 495.749,Z 131.728,A -85,B 0,C 180,E1 -6335.538,E2 -6335.538} C_VEL
LIN {X 0,Y 495.762,Z 131.73,A -85,B 0,C 180,E1 -6338.768,E2 -6338.768} C_VEL
LIN {X 0,Y 495.758,Z 131.721,A -85,B 0,C 180,E1 -6341.781,E2 -6341.781} C_VEL
LIN {X 0,Y 495.74,Z 131.729,A -85,B 0,C 180,E1 -6345.141,E2 -6345.141} C_VEL
LIN {X 0,Y 495.754,Z 131.735,A -85,B 0,C 180,E1 -6348.218,E2 -6348.218} C_VEL
LIN {X 0,Y 495.754,Z 131.729,A -85,B 0,C 180,E1 -6351.408,E2 -6351.408} C_VEL
LIN {X 0,Y 495.752,Z 131.732,A -85,B 0,C 180,E1 -6354.462,E2 -6354.462} C_VEL
LIN {X 0,Y 495.772,Z 131.728,A -85,B 0,C 180,E1 -6357.406,E2 -6357.406} C_VEL
LIN {X 0,Y 495.756,Z 131.73,A -85,B 0,C 180,E1 -6360.713,E2 -6360.713} C_VEL
LIN {X 0,Y 495.095,Z 131.816,A -85,B 0,C 180,E1 -6361.392,E2 -6361.392} C_VEL
LIN {X 0,Y 492.241,Z 132.17,A -85,B 0,C 180,E1 -6362.495,E2 -6362.495} C_VEL
LIN {X 0,Y 489.836,Z 132.472,A -85,B 0,C 180,E1 -6363.383,E2 -6363.383} C_VEL
LIN {X 0,Y 488.82,Z 132.599,A -85,B 0,C 180,E1 -6364.07,E2 -6364.07} C_VEL
LIN {X 0,Y 488.747,Z 132.605,A -85,B 0,C 180,E1 -6364.302,E2 -6364.302} C_VEL
LIN {X 0,Y 488.776,Z 132.697,A -85,B 0,C 180,E1 -6365.304,E2 -6365.304} C_VEL
LIN {X 0,Y 489.617,Z 138.721,A -85,B 0,C 180,E1 -6366.579,E2 -6366.579} C_VEL
LIN {X 0,Y 489.449,Z 149.448,A -85,B 0,C 180,E1 -6368.733,E2 -6368.733} C_VEL
LIN {X 0,Y 491.907,Z 161.964,A -85,B 0,C 180,E1 -6369.028,E2 -6369.028} C_VEL
LIN {X 0,Y 491.325,Z 256.38,A -85,B 0,C 180,E1 -6370.439,E2 -6370.439} C_VEL
LIN {X 0,Y 490.999,Z 270.024,A -85,B 0,C 180,E1 -6370.814,E2 -6370.814} C_VEL
LIN {X 0,Y 490.764,Z 281.671,A -85,B 0,C 180,E1 -6371.294,E2 -6371.294} C_VEL
LIN {X 0,Y 490.413,Z 293.535,A -85,B 0,C 180,E1 -6371.946,E2 -6371.946} C_VEL
LIN {X 0,Y 489.904,Z 305.291,A -85,B 0,C 180,E1 -6372.789,E2 -6372.789} C_VEL
LIN {X 0,Y 489.534,Z 315.824,A -85,B 0,C 180,E1 -6373.742,E2 -6373.742} C_VEL
LIN {X 0,Y 489.22,Z 325.459,A -85,B 0,C 180,E1 -6374.827,E2 -6374.827} C_VEL
LIN {X 0,Y 488.774,Z 334.317,A -85,B 0,C 180,E1 -6376.063,E2 -6376.063} C_VEL
LIN {X 0,Y 488.507,Z 341.592,A -85,B 0,C 180,E1 -6377.326,E2 -6377.326} C_VEL
LIN {X 0,Y 488.354,Z 346.483,A -85,B 0,C 180,E1 -6378.376,E2 -6378.376} C_VEL
LIN {X 0,Y 488.164,Z 351.217,A -85,B 0,C 180,E1 -6379.632,E2 -6379.632} C_VEL
LIN {X 0,Y 488.045,Z 354.825,A -85,B 0,C 180,E1 -6380.885,E2 -6380.885} C_VEL
LIN {X 0,Y 488.01,Z 356.679,A -85,B 0,C 180,E1 -6381.719,E2 -6381.719} C_VEL
LIN {X 0,Y 487.964,Z 358.064,A -85,B 0,C 180,E1 -6382.551,E2 -6382.551} C_VEL
LIN {X 0,Y 488.016,Z 359.211,A -85,B 0,C 180,E1 -6383.558,E2 -6383.558} C_VEL
LIN {X 0,Y 487.918,Z 359.853,A -85,B 0,C 180,E1 -6385.041,E2 -6385.041} C_VEL
LIN {X 0,Y 488.005,Z 359.023,A -85,B 0,C 180,E1 -6386.697,E2 -6386.697} C_VEL
LIN {X 0,Y 488,Z 358.037,A -85,B 0,C 180,E1 -6387.523,E2 -6387.523} C_VEL
LIN {X 0,Y 487.911,Z 356.663,A -85,B 0,C 180,E1 -6388.348,E2 -6388.348} C_VEL
LIN {X 0,Y 488.041,Z 353.767,A -85,B 0,C 180,E1 -6389.587,E2 -6389.587} C_VEL
LIN {X 0,Y 488.06,Z 349.863,A -85,B 0,C 180,E1 -6390.824,E2 -6390.824} C_VEL
LIN {X 0,Y 488.304,Z 344.826,A -85,B 0,C 180,E1 -6392.061,E2 -6392.061} C_VEL
LIN {X 0,Y 488.438,Z 338.508,A -85,B 0,C 180,E1 -6393.299,E2 -6393.299} C_VEL
LIN {X 0,Y 488.707,Z 332.089,A -85,B 0,C 180,E1 -6394.329,E2 -6394.329} C_VEL
LIN {X 0,Y 489.12,Z 324.346,A -85,B 0,C 180,E1 -6395.358,E2 -6395.358} C_VEL
LIN {X 0,Y 489.604,Z 313.853,A -85,B 0,C 180,E1 -6396.49,E2 -6396.49} C_VEL
LIN {X 0,Y 490.056,Z 303.168,A -85,B 0,C 180,E1 -6397.415,E2 -6397.415} C_VEL
LIN {X 0,Y 490.419,Z 292.761,A -85,B 0,C 180,E1 -6398.135,E2 -6398.135} C_VEL
LIN {X 0,Y 490.701,Z 280.535,A -85,B 0,C 180,E1 -6398.792,E2 -6398.792} C_VEL
LIN {X 0,Y 490.955,Z 267.809,A -85,B 0,C 180,E1 -6399.293,E2 -6399.293} C_VEL
LIN {X 0,Y 491.133,Z 254.731,A -85,B 0,C 180,E1 -6399.627,E2 -6399.627} C_VEL
LIN {X 0,Y 491.809,Z 162.413,A -85,B 0,C 180,E1 -6400.985,E2 -6400.985} C_VEL
LIN {X 0,Y 489.293,Z 149.328,A -85,B 0,C 180,E1 -6401.285,E2 -6401.285} C_VEL
LIN {X 0,Y 489.482,Z 137.208,A -85,B 0,C 180,E1 -6403.703,E2 -6403.703} C_VEL
LIN {X 0,Y 488.813,Z 132.6,A -85,B 0,C 180,E1 -6404.678,E2 -6404.678} C_VEL
LIN {X 0,Y 488.75,Z 132.608,A -85,B 0,C 180,E1 -6408.367,E2 -6408.367} C_VEL
LIN {X 0,Y 488.707,Z 132.606,A -85,B 0,C 180,E1 -6411.07,E2 -6411.07} C_VEL
LIN {X 0,Y 488.68,Z 132.612,A -85,B 0,C 180,E1 -6413.745,E2 -6413.745} C_VEL
LIN {X 0,Y 488.79,Z 132.596,A -85,B 0,C 180,E1 -6416.942,E2 -6416.942} C_VEL
LIN {X 0,Y 488.708,Z 132.609,A -85,B 0,C 180,E1 -6420.362,E2 -6420.362} C_VEL
LIN {X 0,Y 488.732,Z 132.606,A -85,B 0,C 180,E1 -6423.483,E2 -6423.483} C_VEL
LIN {X 0,Y 488.678,Z 132.611,A -85,B 0,C 180,E1 -6426.353,E2 -6426.353} C_VEL
LIN {X 0,Y 488.697,Z 132.61,A -85,B 0,C 180,E1 -6429.253,E2 -6429.253} C_VEL
LIN {X 0,Y 488.702,Z 132.613,A -85,B 0,C 180,E1 -6431.599,E2 -6431.599} C_VEL
LIN {X 0,Y 488.695,Z 132.609,A -85,B 0,C 180,E1 -6434.802,E2 -6434.802} C_VEL
LIN {X 0,Y 488.685,Z 132.615,A -85,B 0,C 180,E1 -6437.473,E2 -6437.473} C_VEL
LIN {X 0,Y 488.726,Z 132.608,A -85,B 0,C 180,E1 -6439.676,E2 -6439.676} C_VEL
LIN {X 0,Y 488.67,Z 132.614,A -85,B 0,C 180,E1 -6442.84,E2 -6442.84} C_VEL
LIN {X 0,Y 488.715,Z 132.607,A -85,B 0,C 180,E1 -6445.886,E2 -6445.886} C_VEL
LIN {X 0,Y 488.681,Z 132.613,A -85,B 0,C 180,E1 -6448.819,E2 -6448.819} C_VEL
LIN {X 0,Y 488.731,Z 132.605,A -85,B 0,C 180,E1 -6451.67,E2 -6451.67} C_VEL
LIN {X 0,Y 488.694,Z 132.612,A -85,B 0,C 180,E1 -6454.441,E2 -6454.441} C_VEL
LIN {X 0,Y 488.709,Z 132.61,A -85,B 0,C 180,E1 -6457.152,E2 -6457.152} C_VEL
LIN {X 0,Y 488.711,Z 132.608,A -85,B 0,C 180,E1 -6459.81,E2 -6459.81} C_VEL
LIN {X 0,Y 488.686,Z 132.613,A -85,B 0,C 180,E1 -6462.421,E2 -6462.421} C_VEL
LIN {X 0,Y 488.74,Z 132.606,A -85,B 0,C 180,E1 -6464.999,E2 -6464.999} C_VEL
LIN {X 0,Y 488.792,Z 132.6,A -85,B 0,C 180,E1 -6468.387,E2 -6468.387} C_VEL
LIN {X 0,Y 488.766,Z 132.603,A -85,B 0,C 180,E1 -6471.733,E2 -6471.733} C_VEL
LIN {X 0,Y 488.801,Z 132.599,A -85,B 0,C 180,E1 -6474.223,E2 -6474.223} C_VEL
LIN {X 0,Y 488.929,Z 132.582,A -85,B 0,C 180,E1 -6477.528,E2 -6477.528} C_VEL
LIN {X 0,Y 488.928,Z 132.583,A -85,B 0,C 180,E1 -6480,E2 -6480} C_VEL
LIN {X 0,Y 488.93,Z 132.582,A -85,B 0,C 180,E1 -6482.471,E2 -6482.471} C_VEL
LIN {X 0,Y 488.807,Z 132.598,A -85,B 0,C 180,E1 -6485.776,E2 -6485.776} C_VEL
LIN {X 0,Y 488.766,Z 132.602,A -85,B 0,C 180,E1 -6488.267,E2 -6488.267} C_VEL
LIN {X 0,Y 488.792,Z 132.6,A -85,B 0,C 180,E1 -6491.613,E2 -6491.613} C_VEL
LIN {X 0,Y 488.741,Z 132.606,A -85,B 0,C 180,E1 -6495.001,E2 -6495.001} C_VEL
LIN {X 0,Y 488.733,Z 132.604,A -85,B 0,C 180,E1 -6498.443,E2 -6498.443} C_VEL
LIN {X 0,Y 488.695,Z 132.614,A -85,B 0,C 180,E1 -6501.071,E2 -6501.071} C_VEL
LIN {X 0,Y 488.657,Z 132.615,A -85,B 0,C 180,E1 -6503.747,E2 -6503.747} C_VEL
LIN {X 0,Y 488.736,Z 132.609,A -85,B 0,C 180,E1 -6506.934,E2 -6506.934} C_VEL
LIN {X 0,Y 488.711,Z 132.609,A -85,B 0,C 180,E1 -6509.271,E2 -6509.271} C_VEL
LIN {X 0,Y 488.692,Z 132.609,A -85,B 0,C 180,E1 -6512.148,E2 -6512.148} C_VEL
LIN {X 0,Y 488.705,Z 132.61,A -85,B 0,C 180,E1 -6515.116,E2 -6515.116} C_VEL
LIN {X 0,Y 488.671,Z 132.613,A -85,B 0,C 180,E1 -6518.201,E2 -6518.201} C_VEL
LIN {X 0,Y 488.71,Z 132.61,A -85,B 0,C 180,E1 -6520.346,E2 -6520.346} C_VEL
LIN {X 0,Y 488.677,Z 132.61,A -85,B 0,C 180,E1 -6523.656,E2 -6523.656} C_VEL
LIN {X 0,Y 488.677,Z 132.617,A -85,B 0,C 180,E1 -6526.346,E2 -6526.346} C_VEL
LIN {X 0,Y 488.727,Z 132.605,A -85,B 0,C 180,E1 -6529.678,E2 -6529.678} C_VEL
LIN {X 0,Y 488.674,Z 132.611,A -85,B 0,C 180,E1 -6532.842,E2 -6532.842} C_VEL
LIN {X 0,Y 488.726,Z 132.608,A -85,B 0,C 180,E1 -6535.888,E2 -6535.888} C_VEL
LIN {X 0,Y 488.688,Z 132.608,A -85,B 0,C 180,E1 -6538.821,E2 -6538.821} C_VEL
LIN {X 0,Y 488.742,Z 132.608,A -85,B 0,C 180,E1 -6541.672,E2 -6541.672} C_VEL
LIN {X 0,Y 488.793,Z 132.744,A -85,B 0,C 180,E1 -6544.277,E2 -6544.277} C_VEL
LIN {X 0,Y 490.558,Z 142.115,A -85,B 0,C 180,E1 -6545.903,E2 -6545.903} C_VEL
LIN {X 0,Y 490.401,Z 151.675,A -85,B 0,C 180,E1 -6547.459,E2 -6547.459} C_VEL
LIN {X 0,Y 489.747,Z 172.061,A -85,B 0,C 180,E1 -6550.729,E2 -6550.729} C_VEL
LIN {X 0,Y 489.182,Z 191.242,A -85,B 0,C 180,E1 -6553.758,E2 -6553.758} C_VEL
LIN {X 0,Y 491.586,Z 208.822,A -85,B 0,C 180,E1 -6554.093,E2 -6554.093} C_VEL
LIN {X 0,Y 491.019,Z 299.905,A -85,B 0,C 180,E1 -6555.442,E2 -6555.442} C_VEL
LIN {X 0,Y 490.723,Z 313.173,A -85,B 0,C 180,E1 -6555.804,E2 -6555.804} C_VEL
LIN {X 0,Y 490.321,Z 325.912,A -85,B 0,C 180,E1 -6556.321,E2 -6556.321} C_VEL
LIN {X 0,Y 489.925,Z 337.232,A -85,B 0,C 180,E1 -6556.943,E2 -6556.943} C_VEL
LIN {X 0,Y 489.514,Z 348.929,A -85,B 0,C 180,E1 -6557.775,E2 -6557.775} C_VEL
LIN {X 0,Y 489.099,Z 359.454,A -85,B 0,C 180,E1 -6558.711,E2 -6558.711} C_VEL
LIN {X 0,Y 488.775,Z 368.059,A -85,B 0,C 180,E1 -6559.647,E2 -6559.647} C_VEL
LIN {X 0,Y 488.467,Z 375.993,A -85,B 0,C 180,E1 -6560.686,E2 -6560.686} C_VEL
LIN {X 0,Y 488.239,Z 383.743,A -85,B 0,C 180,E1 -6561.933,E2 -6561.933} C_VEL
LIN {X 0,Y 488.044,Z 390.88,A -85,B 0,C 180,E1 -6563.386,E2 -6563.386} C_VEL
LIN {X 0,Y 488.011,Z 395.633,A -85,B 0,C 180,E1 -6564.63,E2 -6564.63} C_VEL
LIN {X 0,Y 487.93,Z 399.259,A -85,B 0,C 180,E1 -6565.871,E2 -6565.871} C_VEL
LIN {X 0,Y 487.977,Z 401.133,A -85,B 0,C 180,E1 -6566.698,E2 -6566.698} C_VEL
LIN {X 0,Y 487.937,Z 402.535,A -85,B 0,C 180,E1 -6567.524,E2 -6567.524} C_VEL
LIN {X 0,Y 487.893,Z 403.533,A -85,B 0,C 180,E1 -6568.35,E2 -6568.35} C_VEL
LIN {X 0,Y 487.834,Z 404.358,A -85,B 0,C 180,E1 -6570.001,E2 -6570.001} C_VEL
LIN {X 0,Y 487.893,Z 403.533,A -85,B 0,C 180,E1 -6571.652,E2 -6571.652} C_VEL
LIN {X 0,Y 487.937,Z 402.534,A -85,B 0,C 180,E1 -6572.477,E2 -6572.477} C_VEL
LIN {X 0,Y 487.978,Z 401.134,A -85,B 0,C 180,E1 -6573.303,E2 -6573.303} C_VEL
LIN {X 0,Y 487.919,Z 398.184,A -85,B 0,C 180,E1 -6574.545,E2 -6574.545} C_VEL
LIN {X 0,Y 487.996,Z 394.2,A -85,B 0,C 180,E1 -6575.787,E2 -6575.787} C_VEL
LIN {X 0,Y 488.171,Z 388.081,A -85,B 0,C 180,E1 -6577.237,E2 -6577.237} C_VEL
LIN {X 0,Y 488.33,Z 381.393,A -85,B 0,C 180,E1 -6578.484,E2 -6578.484} C_VEL
LIN {X 0,Y 488.608,Z 373.105,A -85,B 0,C 180,E1 -6579.731,E2 -6579.731} C_VEL
LIN {X 0,Y 488.965,Z 364.63,A -85,B 0,C 180,E1 -6580.77,E2 -6580.77} C_VEL
LIN {X 0,Y 489.33,Z 354.166,A -85,B 0,C 180,E1 -6581.811,E2 -6581.811} C_VEL
LIN {X 0,Y 489.739,Z 342.899,A -85,B 0,C 180,E1 -6582.71,E2 -6582.71} C_VEL
LIN {X 0,Y 490.222,Z 330.645,A -85,B 0,C 180,E1 -6583.472,E2 -6583.472} C_VEL
LIN {X 0,Y 490.584,Z 318.437,A -85,B 0,C 180,E1 -6584.043,E2 -6584.043} C_VEL
LIN {X 0,Y 491.001,Z 305.097,A -85,B 0,C 180,E1 -6584.48,E2 -6584.48} C_VEL
LIN {X 0,Y 491.227,Z 291.802,A -85,B 0,C 180,E1 -6584.738,E2 -6584.738} C_VEL
LIN {X 0,Y 491.666,Z 207.683,A -85,B 0,C 180,E1 -6585.977,E2 -6585.977} C_VEL
LIN {X 0,Y 489.24,Z 190.958,A -85,B 0,C 180,E1 -6586.328,E2 -6586.328} C_VEL
LIN {X 0,Y 489.785,Z 172.576,A -85,B 0,C 180,E1 -6589.271,E2 -6589.271} C_VEL
LIN {X 0,Y 490.392,Z 155.138,A -85,B 0,C 180,E1 -6592.099,E2 -6592.099} C_VEL
LIN {X 0,Y 490.789,Z 143.058,A -85,B 0,C 180,E1 -6594.087,E2 -6594.087} C_VEL
LIN {X 0,Y 488.758,Z 132.604,A -85,B 0,C 180,E1 -6595.956,E2 -6595.956} C_VEL
LIN {X 0,Y 488.713,Z 132.61,A -85,B 0,C 180,E1 -6599.271,E2 -6599.271} C_VEL
LIN {X 0,Y 488.706,Z 132.613,A -85,B 0,C 180,E1 -6602.147,E2 -6602.147} C_VEL
LIN {X 0,Y 488.718,Z 132.605,A -85,B 0,C 180,E1 -6605.115,E2 -6605.115} C_VEL
LIN {X 0,Y 488.679,Z 132.61,A -85,B 0,C 180,E1 -6608.2,E2 -6608.2} C_VEL
LIN {X 0,Y 488.721,Z 132.604,A -85,B 0,C 180,E1 -6610.345,E2 -6610.345} C_VEL
LIN {X 0,Y 488.68,Z 132.615,A -85,B 0,C 180,E1 -6613.655,E2 -6613.655} C_VEL
LIN {X 0,Y 488.678,Z 132.61,A -85,B 0,C 180,E1 -6616.344,E2 -6616.344} C_VEL
LIN {X 0,Y 488.704,Z 132.61,A -85,B 0,C 180,E1 -6619.674,E2 -6619.674} C_VEL
LIN {X 0,Y 488.679,Z 132.613,A -85,B 0,C 180,E1 -6622.841,E2 -6622.841} C_VEL
LIN {X 0,Y 488.724,Z 132.604,A -85,B 0,C 180,E1 -6625.887,E2 -6625.887} C_VEL
LIN {X 0,Y 488.686,Z 132.615,A -85,B 0,C 180,E1 -6628.82,E2 -6628.82} C_VEL
LIN {X 0,Y 488.693,Z 132.607,A -85,B 0,C 180,E1 -6631.668,E2 -6631.668} C_VEL
LIN {X 0,Y 488.698,Z 132.612,A -85,B 0,C 180,E1 -6634.959,E2 -6634.959} C_VEL
LIN {X 0,Y 488.688,Z 132.609,A -85,B 0,C 180,E1 -6638.043,E2 -6638.043} C_VEL
LIN {X 0,Y 488.726,Z 132.606,A -85,B 0,C 180,E1 -6640.686,E2 -6640.686} C_VEL
LIN {X 0,Y 488.674,Z 132.61,A -85,B 0,C 180,E1 -6643.284,E2 -6643.284} C_VEL
LIN {X 0,Y 488.711,Z 132.603,A -85,B 0,C 180,E1 -6645.849,E2 -6645.849} C_VEL
LIN {X 0,Y 488.773,Z 132.604,A -85,B 0,C 180,E1 -6648.387,E2 -6648.387} C_VEL
LIN {X 0,Y 488.751,Z 132.598,A -85,B 0,C 180,E1 -6651.733,E2 -6651.733} C_VEL
LIN {X 0,Y 488.807,Z 132.599,A -85,B 0,C 180,E1 -6654.224,E2 -6654.224} C_VEL
LIN {X 0,Y 488.938,Z 132.574,A -85,B 0,C 180,E1 -6657.529,E2 -6657.529} C_VEL
LIN {X 0,Y 488.939,Z 132.583,A -85,B 0,C 180,E1 -6660,E2 -6660} C_VEL
LIN {X 0,Y 488.94,Z 132.573,A -85,B 0,C 180,E1 -6662.472,E2 -6662.472} C_VEL
LIN {X 0,Y 488.81,Z 132.6,A -85,B 0,C 180,E1 -6665.776,E2 -6665.776} C_VEL
LIN {X 0,Y 488.769,Z 132.594,A -85,B 0,C 180,E1 -6668.267,E2 -6668.267} C_VEL
LIN {X 0,Y 488.805,Z 132.6,A -85,B 0,C 180,E1 -6671.613,E2 -6671.613} C_VEL
LIN {X 0,Y 488.753,Z 132.598,A -85,B 0,C 180,E1 -6675.001,E2 -6675.001} C_VEL
LIN {X 0,Y 488.746,Z 132.6,A -85,B 0,C 180,E1 -6678.443,E2 -6678.443} C_VEL
LIN {X 0,Y 488.707,Z 132.61,A -85,B 0,C 180,E1 -6681.071,E2 -6681.071} C_VEL
LIN {X 0,Y 488.669,Z 132.608,A -85,B 0,C 180,E1 -6683.747,E2 -6683.747} C_VEL
LIN {X 0,Y 488.726,Z 132.611,A -85,B 0,C 180,E1 -6686.928,E2 -6686.928} C_VEL
LIN {X 0,Y 488.723,Z 132.604,A -85,B 0,C 180,E1 -6690.22,E2 -6690.22} C_VEL
LIN {X 0,Y 488.731,Z 132.603,A -85,B 0,C 180,E1 -6693.483,E2 -6693.483} C_VEL
LIN {X 0,Y 488.684,Z 132.612,A -85,B 0,C 180,E1 -6696.355,E2 -6696.355} C_VEL
LIN {X 0,Y 488.7,Z 132.605,A -85,B 0,C 180,E1 -6699.255,E2 -6699.255} C_VEL
LIN {X 0,Y 488.709,Z 132.598,A -85,B 0,C 180,E1 -6701.6,E2 -6701.6} C_VEL
LIN {X 0,Y 488.704,Z 132.608,A -85,B 0,C 180,E1 -6704.803,E2 -6704.803} C_VEL
LIN {X 0,Y 488.691,Z 132.608,A -85,B 0,C 180,E1 -6707.474,E2 -6707.474} C_VEL
LIN {X 0,Y 488.705,Z 132.608,A -85,B 0,C 180,E1 -6710.746,E2 -6710.746} C_VEL
LIN {X 0,Y 488.681,Z 132.615,A -85,B 0,C 180,E1 -6713.868,E2 -6713.868} C_VEL
LIN {X 0,Y 488.743,Z 132.602,A -85,B 0,C 180,E1 -6716.877,E2 -6716.877} C_VEL
LIN {X 0,Y 488.728,Z 132.61,A -85,B 0,C 180,E1 -6719.781,E2 -6719.781} C_VEL
LIN {X 0,Y 488.796,Z 132.599,A -85,B 0,C 180,E1 -6723.057,E2 -6723.057} C_VEL
LIN {X 0,Y 488.747,Z 132.605,A -85,B 0,C 180,E1 -6724.302,E2 -6724.302} C_VEL
LIN {X 0,Y 488.485,Z 132.968,A -85,B 0,C 180,E1 -6724.757,E2 -6724.757} C_VEL
LIN {X 0,Y 487.339,Z 134.587,A -85,B 0,C 180,E1 -6725.41,E2 -6725.41} C_VEL
LIN {X 0,Y 485.747,Z 137.073,A -85,B 0,C 180,E1 -6726.021,E2 -6726.021} C_VEL
LIN {X 0,Y 482.901,Z 143.464,A -85,B 0,C 180,E1 -6727.219,E2 -6727.219} C_VEL
LIN {X 0,Y 482.587,Z 145.555,A -85,B 0,C 180,E1 -6727.631,E2 -6727.631} C_VEL
LIN {X 0,Y 482.492,Z 149.775,A -85,B 0,C 180,E1 -6728.48,E2 -6728.48} C_VEL
LIN {X 0,Y 485.142,Z 163.206,A -85,B 0,C 180,E1 -6728.796,E2 -6728.796} C_VEL
LIN {X 0,Y 484.529,Z 256.483,A -85,B 0,C 180,E1 -6730.208,E2 -6730.208} C_VEL
LIN {X 0,Y 484.222,Z 269.625,A -85,B 0,C 180,E1 -6730.569,E2 -6730.569} C_VEL
LIN {X 0,Y 483.927,Z 281.566,A -85,B 0,C 180,E1 -6731.059,E2 -6731.059} C_VEL
LIN {X 0,Y 483.587,Z 292.904,A -85,B 0,C 180,E1 -6731.682,E2 -6731.682} C_VEL
LIN {X 0,Y 483.107,Z 303.584,A -85,B 0,C 180,E1 -6732.43,E2 -6732.43} C_VEL
LIN {X 0,Y 482.733,Z 314.469,A -85,B 0,C 180,E1 -6733.398,E2 -6733.398} C_VEL
LIN {X 0,Y 482.298,Z 324.162,A -85,B 0,C 180,E1 -6734.462,E2 -6734.462} C_VEL
LIN {X 0,Y 481.855,Z 332.896,A -85,B 0,C 180,E1 -6735.643,E2 -6735.643} C_VEL
LIN {X 0,Y 481.534,Z 340.476,A -85,B 0,C 180,E1 -6736.925,E2 -6736.925} C_VEL
LIN {X 0,Y 481.342,Z 346.547,A -85,B 0,C 180,E1 -6738.204,E2 -6738.204} C_VEL
LIN {X 0,Y 481.115,Z 351.336,A -85,B 0,C 180,E1 -6739.478,E2 -6739.478} C_VEL
LIN {X 0,Y 480.974,Z 354.995,A -85,B 0,C 180,E1 -6740.75,E2 -6740.75} C_VEL
LIN {X 0,Y 480.941,Z 356.879,A -85,B 0,C 180,E1 -6741.597,E2 -6741.597} C_VEL
LIN {X 0,Y 480.899,Z 358.307,A -85,B 0,C 180,E1 -6742.441,E2 -6742.441} C_VEL
LIN {X 0,Y 480.933,Z 359.577,A -85,B 0,C 180,E1 -6743.569,E2 -6743.569} C_VEL
LIN {X 0,Y 480.847,Z 360.171,A -85,B 0,C 180,E1 -6744.968,E2 -6744.968} C_VEL
LIN {X 0,Y 480.86,Z 359.989,A -85,B 0,C 180,E1 -6745.809,E2 -6745.809} C_VEL
LIN {X 0,Y 480.926,Z 359.404,A -85,B 0,C 180,E1 -6746.648,E2 -6746.648} C_VEL
LIN {X 0,Y 480.908,Z 358.442,A -85,B 0,C 180,E1 -6747.486,E2 -6747.486} C_VEL
LIN {X 0,Y 480.842,Z 357.098,A -85,B 0,C 180,E1 -6748.324,E2 -6748.324} C_VEL
LIN {X 0,Y 480.943,Z 354.245,A -85,B 0,C 180,E1 -6749.581,E2 -6749.581} C_VEL
LIN {X 0,Y 480.981,Z 350.391,A -85,B 0,C 180,E1 -6750.836,E2 -6750.836} C_VEL
LIN {X 0,Y 481.242,Z 345.41,A -85,B 0,C 180,E1 -6752.092,E2 -6752.092} C_VEL
LIN {X 0,Y 481.384,Z 339.176,A -85,B 0,C 180,E1 -6753.347,E2 -6753.347} C_VEL
LIN {X 0,Y 481.672,Z 332.809,A -85,B 0,C 180,E1 -6754.392,E2 -6754.392} C_VEL
LIN {X 0,Y 482.104,Z 325.154,A -85,B 0,C 180,E1 -6755.436,E2 -6755.436} C_VEL
LIN {X 0,Y 482.614,Z 314.769,A -85,B 0,C 180,E1 -6756.584,E2 -6756.584} C_VEL
LIN {X 0,Y 483.087,Z 304.207,A -85,B 0,C 180,E1 -6757.523,E2 -6757.523} C_VEL
LIN {X 0,Y 483.472,Z 294,A -85,B 0,C 180,E1 -6758.252,E2 -6758.252} C_VEL
LIN {X 0,Y 483.735,Z 283.634,A -85,B 0,C 180,E1 -6758.845,E2 -6758.845} C_VEL
LIN {X 0,Y 484.003,Z 270.557,A -85,B 0,C 180,E1 -6759.401,E2 -6759.401} C_VEL
LIN {X 0,Y 484.22,Z 257.801,A -85,B 0,C 180,E1 -6759.766,E2 -6759.766} C_VEL
LIN {X 0,Y 484.57,Z 219.105,A -85,B 0,C 180,E1 -6760.365,E2 -6760.365} C_VEL
LIN {X 0,Y 484.874,Z 162.482,A -85,B 0,C 180,E1 -6761.207,E2 -6761.207} C_VEL
LIN {X 0,Y 482.33,Z 149.639,A -85,B 0,C 180,E1 -6761.503,E2 -6761.503} C_VEL
LIN {X 0,Y 482.512,Z 138.752,A -85,B 0,C 180,E1 -6763.69,E2 -6763.69} C_VEL
LIN {X 0,Y 481.776,Z 133.476,A -85,B 0,C 180,E1 -6764.843,E2 -6764.843} C_VEL
LIN {X 0,Y 481.7,Z 133.484,A -85,B 0,C 180,E1 -6768.494,E2 -6768.494} C_VEL
LIN {X 0,Y 481.646,Z 133.485,A -85,B 0,C 180,E1 -6771.394,E2 -6771.394} C_VEL
LIN {X 0,Y 481.661,Z 133.49,A -85,B 0,C 180,E1 -6774.113,E2 -6774.113} C_VEL
LIN {X 0,Y 481.744,Z 133.473,A -85,B 0,C 180,E1 -6777.138,E2 -6777.138} C_VEL
LIN {X 0,Y 481.676,Z 133.485,A -85,B 0,C 180,E1 -6779.74,E2 -6779.74} C_VEL
LIN {X 0,Y 481.669,Z 133.483,A -85,B 0,C 180,E1 -6782.673,E2 -6782.673} C_VEL
LIN {X 0,Y 481.633,Z 133.492,A -85,B 0,C 180,E1 -6785.708,E2 -6785.708} C_VEL
LIN {X 0,Y 481.667,Z 133.484,A -85,B 0,C 180,E1 -6788.858,E2 -6788.858} C_VEL
LIN {X 0,Y 481.647,Z 133.49,A -85,B 0,C 180,E1 -6791.912,E2 -6791.912} C_VEL
LIN {X 0,Y 481.649,Z 133.486,A -85,B 0,C 180,E1 -6794.457,E2 -6794.457} C_VEL
LIN {X 0,Y 481.64,Z 133.49,A -85,B 0,C 180,E1 -6797.838,E2 -6797.838} C_VEL
LIN {X 0,Y 481.653,Z 133.487,A -85,B 0,C 180,E1 -6800.653,E2 -6800.653} C_VEL
LIN {X 0,Y 481.619,Z 133.496,A -85,B 0,C 180,E1 -6803.375,E2 -6803.375} C_VEL
LIN {X 0,Y 481.667,Z 133.485,A -85,B 0,C 180,E1 -6806.326,E2 -6806.326} C_VEL
LIN {X 0,Y 481.64,Z 133.491,A -85,B 0,C 180,E1 -6809.417,E2 -6809.417} C_VEL
LIN {X 0,Y 481.681,Z 133.484,A -85,B 0,C 180,E1 -6812.167,E2 -6812.167} C_VEL
LIN {X 0,Y 481.663,Z 133.489,A -85,B 0,C 180,E1 -6814.967,E2 -6814.967} C_VEL
LIN {X 0,Y 481.636,Z 133.489,A -85,B 0,C 180,E1 -6817.704,E2 -6817.704} C_VEL
LIN {X 0,Y 481.688,Z 133.484,A -85,B 0,C 180,E1 -6820.392,E2 -6820.392} C_VEL
LIN {X 0,Y 481.648,Z 133.49,A -85,B 0,C 180,E1 -6823.032,E2 -6823.032} C_VEL
LIN {X 0,Y 481.662,Z 133.486,A -85,B 0,C 180,E1 -6825.638,E2 -6825.638} C_VEL
LIN {X 0,Y 481.738,Z 133.478,A -85,B 0,C 180,E1 -6828.215,E2 -6828.215} C_VEL
LIN {X 0,Y 481.722,Z 133.479,A -85,B 0,C 180,E1 -6831.611,E2 -6831.611} C_VEL
LIN {X 0,Y 481.762,Z 133.475,A -85,B 0,C 180,E1 -6834.139,E2 -6834.139} C_VEL
LIN {X 0,Y 481.894,Z 133.458,A -85,B 0,C 180,E1 -6837.492,E2 -6837.492} C_VEL
LIN {X 0,Y 481.897,Z 133.458,A -85,B 0,C 180,E1 -6840,E2 -6840} C_VEL
LIN {X 0,Y 481.895,Z 133.458,A -85,B 0,C 180,E1 -6842.508,E2 -6842.508} C_VEL
LIN {X 0,Y 481.768,Z 133.474,A -85,B 0,C 180,E1 -6845.861,E2 -6845.861} C_VEL
LIN {X 0,Y 481.722,Z 133.479,A -85,B 0,C 180,E1 -6848.389,E2 -6848.389} C_VEL
LIN {X 0,Y 481.738,Z 133.478,A -85,B 0,C 180,E1 -6851.785,E2 -6851.785} C_VEL
LIN {X 0,Y 481.725,Z 133.482,A -85,B 0,C 180,E1 -6855.225,E2 -6855.225} C_VEL
LIN {X 0,Y 481.695,Z 133.482,A -85,B 0,C 180,E1 -6858.722,E2 -6858.722} C_VEL
LIN {X 0,Y 481.633,Z 133.491,A -85,B 0,C 180,E1 -6861.395,E2 -6861.395} C_VEL
LIN {X 0,Y 481.637,Z 133.488,A -85,B 0,C 180,E1 -6864.115,E2 -6864.115} C_VEL
LIN {X 0,Y 481.704,Z 133.483,A -85,B 0,C 180,E1 -6867.132,E2 -6867.132} C_VEL
LIN {X 0,Y 481.667,Z 133.485,A -85,B 0,C 180,E1 -6869.742,E2 -6869.742} C_VEL
LIN {X 0,Y 481.66,Z 133.49,A -85,B 0,C 180,E1 -6872.675,E2 -6872.675} C_VEL
LIN {X 0,Y 481.626,Z 133.489,A -85,B 0,C 180,E1 -6875.711,E2 -6875.711} C_VEL
LIN {X 0,Y 481.662,Z 133.488,A -85,B 0,C 180,E1 -6878.86,E2 -6878.86} C_VEL
LIN {X 0,Y 481.644,Z 133.487,A -85,B 0,C 180,E1 -6881.914,E2 -6881.914} C_VEL
LIN {X 0,Y 481.647,Z 133.492,A -85,B 0,C 180,E1 -6884.459,E2 -6884.459} C_VEL
LIN {X 0,Y 481.641,Z 133.488,A -85,B 0,C 180,E1 -6887.84,E2 -6887.84} C_VEL
LIN {X 0,Y 481.675,Z 133.485,A -85,B 0,C 180,E1 -6890.652,E2 -6890.652} C_VEL
LIN {X 0,Y 481.622,Z 133.489,A -85,B 0,C 180,E1 -6893.377,E2 -6893.377} C_VEL
LIN {X 0,Y 481.706,Z 133.482,A -85,B 0,C 180,E1 -6896.331,E2 -6896.331} C_VEL
LIN {X 0,Y 481.647,Z 133.486,A -85,B 0,C 180,E1 -6899.419,E2 -6899.419} C_VEL
LIN {X 0,Y 481.697,Z 133.485,A -85,B 0,C 180,E1 -6902.169,E2 -6902.169} C_VEL
LIN {X 0,Y 481.744,Z 133.573,A -85,B 0,C 180,E1 -6904.092,E2 -6904.092} C_VEL
LIN {X 0,Y 483.693,Z 144.403,A -85,B 0,C 180,E1 -6905.995,E2 -6905.995} C_VEL
LIN {X 0,Y 483.076,Z 163.48,A -85,B 0,C 180,E1 -6909.12,E2 -6909.12} C_VEL
LIN {X 0,Y 482.429,Z 182.46,A -85,B 0,C 180,E1 -6912.187,E2 -6912.187} C_VEL
LIN {X 0,Y 482.174,Z 190.808,A -85,B 0,C 180,E1 -6913.527,E2 -6913.527} C_VEL
LIN {X 0,Y 484.736,Z 209.462,A -85,B 0,C 180,E1 -6913.892,E2 -6913.892} C_VEL
LIN {X 0,Y 484.127,Z 300.112,A -85,B 0,C 180,E1 -6915.257,E2 -6915.257} C_VEL
LIN {X 0,Y 483.841,Z 312.444,A -85,B 0,C 180,E1 -6915.598,E2 -6915.598} C_VEL
LIN {X 0,Y 483.396,Z 325.293,A -85,B 0,C 180,E1 -6916.121,E2 -6916.121} C_VEL
LIN {X 0,Y 482.972,Z 336.705,A -85,B 0,C 180,E1 -6916.752,E2 -6916.752} C_VEL
LIN {X 0,Y 482.567,Z 347.5,A -85,B 0,C 180,E1 -6917.519,E2 -6917.519} C_VEL
LIN {X 0,Y 482.108,Z 359.004,A -85,B 0,C 180,E1 -6918.545,E2 -6918.545} C_VEL
LIN {X 0,Y 481.733,Z 367.631,A -85,B 0,C 180,E1 -6919.494,E2 -6919.494} C_VEL
LIN {X 0,Y 481.433,Z 375.589,A -85,B 0,C 180,E1 -6920.548,E2 -6920.548} C_VEL
LIN {X 0,Y 481.163,Z 383.362,A -85,B 0,C 180,E1 -6921.814,E2 -6921.814} C_VEL
LIN {X 0,Y 480.963,Z 390.513,A -85,B 0,C 180,E1 -6923.288,E2 -6923.288} C_VEL
LIN {X 0,Y 480.922,Z 395.276,A -85,B 0,C 180,E1 -6924.55,E2 -6924.55} C_VEL
LIN {X 0,Y 480.83,Z 398.912,A -85,B 0,C 180,E1 -6925.81,E2 -6925.81} C_VEL
LIN {X 0,Y 480.9,Z 400.793,A -85,B 0,C 180,E1 -6926.65,E2 -6926.65} C_VEL
LIN {X 0,Y 480.849,Z 402.2,A -85,B 0,C 180,E1 -6927.488,E2 -6927.488} C_VEL
LIN {X 0,Y 480.824,Z 403.203,A -85,B 0,C 180,E1 -6928.326,E2 -6928.326} C_VEL
LIN {X 0,Y 480.757,Z 404.035,A -85,B 0,C 180,E1 -6930.001,E2 -6930.001} C_VEL
LIN {X 0,Y 480.824,Z 403.218,A -85,B 0,C 180,E1 -6931.676,E2 -6931.676} C_VEL
LIN {X 0,Y 480.85,Z 402.222,A -85,B 0,C 180,E1 -6932.514,E2 -6932.514} C_VEL
LIN {X 0,Y 480.9,Z 400.827,A -85,B 0,C 180,E1 -6933.352,E2 -6933.352} C_VEL
LIN {X 0,Y 480.837,Z 397.883,A -85,B 0,C 180,E1 -6934.612,E2 -6934.612} C_VEL
LIN {X 0,Y 480.895,Z 393.907,A -85,B 0,C 180,E1 -6935.872,E2 -6935.872} C_VEL
LIN {X 0,Y 481.095,Z 387.804,A -85,B 0,C 180,E1 -6937.344,E2 -6937.344} C_VEL
LIN {X 0,Y 481.274,Z 381.132,A -85,B 0,C 180,E1 -6938.609,E2 -6938.609} C_VEL
LIN {X 0,Y 481.544,Z 372.862,A -85,B 0,C 180,E1 -6939.875,E2 -6939.875} C_VEL
LIN {X 0,Y 481.979,Z 364.412,A -85,B 0,C 180,E1 -6940.928,E2 -6940.928} C_VEL
LIN {X 0,Y 482.354,Z 354.179,A -85,B 0,C 180,E1 -6941.966,E2 -6941.966} C_VEL
LIN {X 0,Y 482.727,Z 343.976,A -85,B 0,C 180,E1 -6942.807,E2 -6942.807} C_VEL
LIN {X 0,Y 483.222,Z 332.435,A -85,B 0,C 180,E1 -6943.564,E2 -6943.564} C_VEL
LIN {X 0,Y 483.659,Z 319.766,A -85,B 0,C 180,E1 -6944.195,E2 -6944.195} C_VEL
LIN {X 0,Y 484.099,Z 307.106,A -85,B 0,C 180,E1 -6944.638,E2 -6944.638} C_VEL
LIN {X 0,Y 484.37,Z 294.129,A -85,B 0,C 180,E1 -6944.925,E2 -6944.925} C_VEL
LIN {X 0,Y 484.892,Z 208.409,A -85,B 0,C 180,E1 -6946.207,E2 -6946.207} C_VEL
LIN {X 0,Y 482.235,Z 190.602,A -85,B 0,C 180,E1 -6946.593,E2 -6946.593} C_VEL
LIN {X 0,Y 482.854,Z 172.365,A -85,B 0,C 180,E1 -6949.559,E2 -6949.559} C_VEL
LIN {X 0,Y 483.541,Z 154.942,A -85,B 0,C 180,E1 -6952.429,E2 -6952.429} C_VEL
LIN {X 0,Y 483.943,Z 145.556,A -85,B 0,C 180,E1 -6953.994,E2 -6953.994} C_VEL
LIN {X 0,Y 482.348,Z 136.539,A -85,B 0,C 180,E1 -6955.615,E2 -6955.615} C_VEL
LIN {X 0,Y 481.693,Z 133.485,A -85,B 0,C 180,E1 -6956.191,E2 -6956.191} C_VEL
LIN {X 0,Y 481.657,Z 133.489,A -85,B 0,C 180,E1 -6958.898,E2 -6958.898} C_VEL
LIN {X 0,Y 481.66,Z 133.491,A -85,B 0,C 180,E1 -6962.189,E2 -6962.189} C_VEL
LIN {X 0,Y 481.69,Z 133.48,A -85,B 0,C 180,E1 -6964.682,E2 -6964.682} C_VEL
LIN {X 0,Y 481.653,Z 133.488,A -85,B 0,C 180,E1 -6968.007,E2 -6968.007} C_VEL
LIN {X 0,Y 481.651,Z 133.486,A -85,B 0,C 180,E1 -6971.043,E2 -6971.043} C_VEL
LIN {X 0,Y 481.656,Z 133.484,A -85,B 0,C 180,E1 -6974.458,E2 -6974.458} C_VEL
LIN {X 0,Y 481.641,Z 133.489,A -85,B 0,C 180,E1 -6977.838,E2 -6977.838} C_VEL
LIN {X 0,Y 481.667,Z 133.489,A -85,B 0,C 180,E1 -6981.14,E2 -6981.14} C_VEL
LIN {X 0,Y 481.636,Z 133.487,A -85,B 0,C 180,E1 -6984.29,E2 -6984.29} C_VEL
LIN {X 0,Y 481.67,Z 133.487,A -85,B 0,C 180,E1 -6987.326,E2 -6987.326} C_VEL
LIN {X 0,Y 481.665,Z 133.484,A -85,B 0,C 180,E1 -6990.258,E2 -6990.258} C_VEL
LIN {X 0,Y 481.66,Z 133.487,A -85,B 0,C 180,E1 -6993.107,E2 -6993.107} C_VEL
LIN {X 0,Y 481.646,Z 133.485,A -85,B 0,C 180,E1 -6995.885,E2 -6995.885} C_VEL
LIN {X 0,Y 481.688,Z 133.48,A -85,B 0,C 180,E1 -6999.032,E2 -6999.032} C_VEL
LIN {X 0,Y 481.665,Z 133.484,A -85,B 0,C 180,E1 -7002.157,E2 -7002.157} C_VEL
LIN {X 0,Y 481.727,Z 133.474,A -85,B 0,C 180,E1 -7004.775,E2 -7004.775} C_VEL
LIN {X 0,Y 481.724,Z 133.481,A -85,B 0,C 180,E1 -7008.214,E2 -7008.214} C_VEL
LIN {X 0,Y 481.71,Z 133.474,A -85,B 0,C 180,E1 -7011.611,E2 -7011.611} C_VEL
LIN {X 0,Y 481.769,Z 133.477,A -85,B 0,C 180,E1 -7014.139,E2 -7014.139} C_VEL
LIN {X 0,Y 481.903,Z 133.45,A -85,B 0,C 180,E1 -7017.493,E2 -7017.493} C_VEL
LIN {X 0,Y 481.909,Z 133.459,A -85,B 0,C 180,E1 -7020,E2 -7020} C_VEL
LIN {X 0,Y 481.905,Z 133.448,A -85,B 0,C 180,E1 -7022.508,E2 -7022.508} C_VEL
LIN {X 0,Y 481.771,Z 133.475,A -85,B 0,C 180,E1 -7025.861,E2 -7025.861} C_VEL
LIN {X 0,Y 481.728,Z 133.47,A -85,B 0,C 180,E1 -7028.389,E2 -7028.389} C_VEL
LIN {X 0,Y 481.751,Z 133.476,A -85,B 0,C 180,E1 -7031.785,E2 -7031.785} C_VEL
LIN {X 0,Y 481.738,Z 133.475,A -85,B 0,C 180,E1 -7035.225,E2 -7035.225} C_VEL
LIN {X 0,Y 481.707,Z 133.478,A -85,B 0,C 180,E1 -7038.722,E2 -7038.722} C_VEL
LIN {X 0,Y 481.646,Z 133.49,A -85,B 0,C 180,E1 -7041.395,E2 -7041.395} C_VEL
LIN {X 0,Y 481.649,Z 133.481,A -85,B 0,C 180,E1 -7044.115,E2 -7044.115} C_VEL
LIN {X 0,Y 481.696,Z 133.484,A -85,B 0,C 180,E1 -7047.127,E2 -7047.127} C_VEL
LIN {X 0,Y 481.673,Z 133.481,A -85,B 0,C 180,E1 -7049.742,E2 -7049.742} C_VEL
LIN {X 0,Y 481.672,Z 133.486,A -85,B 0,C 180,E1 -7052.674,E2 -7052.674} C_VEL
LIN {X 0,Y 481.638,Z 133.485,A -85,B 0,C 180,E1 -7055.71,E2 -7055.71} C_VEL
LIN {X 0,Y 481.67,Z 133.484,A -85,B 0,C 180,E1 -7058.86,E2 -7058.86} C_VEL
LIN {X 0,Y 481.655,Z 133.478,A -85,B 0,C 180,E1 -7061.913,E2 -7061.913} C_VEL
LIN {X 0,Y 481.658,Z 133.489,A -85,B 0,C 180,E1 -7064.458,E2 -7064.458} C_VEL
LIN {X 0,Y 481.646,Z 133.488,A -85,B 0,C 180,E1 -7067.839,E2 -7067.839} C_VEL
LIN {X 0,Y 481.664,Z 133.485,A -85,B 0,C 180,E1 -7070.654,E2 -7070.654} C_VEL
LIN {X 0,Y 481.631,Z 133.488,A -85,B 0,C 180,E1 -7073.376,E2 -7073.376} C_VEL
LIN {X 0,Y 481.714,Z 133.481,A -85,B 0,C 180,E1 -7076.33,E2 -7076.33} C_VEL
LIN {X 0,Y 481.655,Z 133.488,A -85,B 0,C 180,E1 -7079.417,E2 -7079.417} C_VEL
LIN {X 0,Y 481.702,Z 133.485,A -85,B 0,C 180,E1 -7082.168,E2 -7082.168} C_VEL
LIN {X 0,Y 481.756,Z 133.668,A -85,B 0,C 180,E1 -7085.144,E2 -7085.144} C_VEL
LIN {X 0,Y 482.689,Z 140.158,A -85,B 0,C 180,E1 -7086.533,E2 -7086.533} C_VEL
LIN {X 0,Y 482.587,Z 145.555,A -85,B 0,C 180,E1 -7087.631,E2 -7087.631} C_VEL
LIN {X 0,Y 482.353,Z 148.029,A -85,B 0,C 180,E1 -7087.976,E2 -7087.976} C_VEL
LIN {X 0,Y 481.704,Z 152.084,A -85,B 0,C 180,E1 -7088.283,E2 -7088.283} C_VEL
LIN {X 0,Y 480.849,Z 156.694,A -85,B 0,C 180,E1 -7088.474,E2 -7088.474} C_VEL
LIN {X 0,Y 479.647,Z 162.777,A -85,B 0,C 180,E1 -7088.579,E2 -7088.579} C_VEL
LIN {X 0,Y 478.514,Z 171.233,A -85,B 0,C 180,E1 -7088.664,E2 -7088.664} C_VEL
LIN {X 0,Y 478.376,Z 175.483,A -85,B 0,C 180,E1 -7088.726,E2 -7088.726} C_VEL
LIN {X 0,Y 477.691,Z 257.824,A -85,B 0,C 180,E1 -7089.997,E2 -7089.997} C_VEL
LIN {X 0,Y 477.354,Z 271.13,A -85,B 0,C 180,E1 -7090.381,E2 -7090.381} C_VEL
LIN {X 0,Y 477.071,Z 282.883,A -85,B 0,C 180,E1 -7090.884,E2 -7090.884} C_VEL
LIN {X 0,Y 476.684,Z 294.039,A -85,B 0,C 180,E1 -7091.519,E2 -7091.519} C_VEL
LIN {X 0,Y 476.102,Z 305.816,A -85,B 0,C 180,E1 -7092.385,E2 -7092.385} C_VEL
LIN {X 0,Y 475.683,Z 316.364,A -85,B 0,C 180,E1 -7093.365,E2 -7093.365} C_VEL
LIN {X 0,Y 475.315,Z 325.547,A -85,B 0,C 180,E1 -7094.419,E2 -7094.419} C_VEL
LIN {X 0,Y 474.836,Z 334.209,A -85,B 0,C 180,E1 -7095.645,E2 -7095.645} C_VEL
LIN {X 0,Y 474.485,Z 341.612,A -85,B 0,C 180,E1 -7096.945,E2 -7096.945} C_VEL
LIN {X 0,Y 474.192,Z 348.386,A -85,B 0,C 180,E1 -7098.458,E2 -7098.458} C_VEL
LIN {X 0,Y 473.991,Z 352.832,A -85,B 0,C 180,E1 -7099.75,E2 -7099.75} C_VEL
LIN {X 0,Y 473.912,Z 355.171,A -85,B 0,C 180,E1 -7100.611,E2 -7100.611} C_VEL
LIN {X 0,Y 473.87,Z 357.078,A -85,B 0,C 180,E1 -7101.47,E2 -7101.47} C_VEL
LIN {X 0,Y 473.828,Z 358.552,A -85,B 0,C 180,E1 -7102.328,E2 -7102.328} C_VEL
LIN {X 0,Y 473.863,Z 359.931,A -85,B 0,C 180,E1 -7103.566,E2 -7103.566} C_VEL
LIN {X 0,Y 473.778,Z 360.483,A -85,B 0,C 180,E1 -7104.893,E2 -7104.893} C_VEL
LIN {X 0,Y 473.765,Z 360.346,A -85,B 0,C 180,E1 -7105.746,E2 -7105.746} C_VEL
LIN {X 0,Y 473.849,Z 359.783,A -85,B 0,C 180,E1 -7106.598,E2 -7106.598} C_VEL
LIN {X 0,Y 473.776,Z 357.52,A -85,B 0,C 180,E1 -7108.299,E2 -7108.299} C_VEL
LIN {X 0,Y 473.847,Z 354.716,A -85,B 0,C 180,E1 -7109.574,E2 -7109.574} C_VEL
LIN {X 0,Y 473.901,Z 350.91,A -85,B 0,C 180,E1 -7110.849,E2 -7110.849} C_VEL
LIN {X 0,Y 474.182,Z 345.981,A -85,B 0,C 180,E1 -7112.123,E2 -7112.123} C_VEL
LIN {X 0,Y 474.332,Z 339.814,A -85,B 0,C 180,E1 -7113.397,E2 -7113.397} C_VEL
LIN {X 0,Y 474.639,Z 333.499,A -85,B 0,C 180,E1 -7114.458,E2 -7114.458} C_VEL
LIN {X 0,Y 475.092,Z 325.92,A -85,B 0,C 180,E1 -7115.517,E2 -7115.517} C_VEL
LIN {X 0,Y 475.56,Z 316.724,A -85,B 0,C 180,E1 -7116.576,E2 -7116.576} C_VEL
LIN {X 0,Y 476.044,Z 306.499,A -85,B 0,C 180,E1 -7117.528,E2 -7117.528} C_VEL
LIN {X 0,Y 476.527,Z 295.163,A -85,B 0,C 180,E1 -7118.373,E2 -7118.373} C_VEL
LIN {X 0,Y 476.866,Z 282.788,A -85,B 0,C 180,E1 -7119.089,E2 -7119.089} C_VEL
LIN {X 0,Y 477.135,Z 270.232,A -85,B 0,C 180,E1 -7119.618,E2 -7119.618} C_VEL
LIN {X 0,Y 477.373,Z 257.144,A -85,B 0,C 180,E1 -7119.987,E2 -7119.987} C_VEL
LIN {X 0,Y 478.006,Z 163.224,A -85,B 0,C 180,E1 -7121.421,E2 -7121.421} C_VEL
LIN {X 0,Y 475.399,Z 149.94,A -85,B 0,C 180,E1 -7121.727,E2 -7121.727} C_VEL
LIN {X 0,Y 475.496,Z 139.263,A -85,B 0,C 180,E1 -7123.896,E2 -7123.896} C_VEL
LIN {X 0,Y 474.747,Z 134.351,A -85,B 0,C 180,E1 -7124.959,E2 -7124.959} C_VEL
LIN {X 0,Y 474.66,Z 134.359,A -85,B 0,C 180,E1 -7128.627,E2 -7128.627} C_VEL
LIN {X 0,Y 474.635,Z 134.359,A -85,B 0,C 180,E1 -7131.115,E2 -7131.115} C_VEL
LIN {X 0,Y 474.64,Z 134.362,A -85,B 0,C 180,E1 -7134.493,E2 -7134.493} C_VEL
LIN {X 0,Y 474.679,Z 134.354,A -85,B 0,C 180,E1 -7137.333,E2 -7137.333} C_VEL
LIN {X 0,Y 474.602,Z 134.364,A -85,B 0,C 180,E1 -7140.809,E2 -7140.809} C_VEL
LIN {X 0,Y 474.635,Z 134.365,A -85,B 0,C 180,E1 -7143.983,E2 -7143.983} C_VEL
LIN {X 0,Y 474.568,Z 134.368,A -85,B 0,C 180,E1 -7146.898,E2 -7146.898} C_VEL
LIN {X 0,Y 474.623,Z 134.366,A -85,B 0,C 180,E1 -7149.646,E2 -7149.646} C_VEL
LIN {X 0,Y 474.609,Z 134.364,A -85,B 0,C 180,E1 -7152.933,E2 -7152.933} C_VEL
LIN {X 0,Y 474.599,Z 134.367,A -85,B 0,C 180,E1 -7155.893,E2 -7155.893} C_VEL
LIN {X 0,Y 474.62,Z 134.364,A -85,B 0,C 180,E1 -7159.04,E2 -7159.04} C_VEL
LIN {X 0,Y 474.602,Z 134.367,A -85,B 0,C 180,E1 -7161.703,E2 -7161.703} C_VEL
LIN {X 0,Y 474.614,Z 134.365,A -85,B 0,C 180,E1 -7164.724,E2 -7164.724} C_VEL
LIN {X 0,Y 474.625,Z 134.363,A -85,B 0,C 180,E1 -7167.787,E2 -7167.787} C_VEL
LIN {X 0,Y 474.612,Z 134.366,A -85,B 0,C 180,E1 -7170.884,E2 -7170.884} C_VEL
LIN {X 0,Y 474.615,Z 134.364,A -85,B 0,C 180,E1 -7173.625,E2 -7173.625} C_VEL
LIN {X 0,Y 474.623,Z 134.364,A -85,B 0,C 180,E1 -7176.641,E2 -7176.641} C_VEL
LIN {X 0,Y 474.639,Z 134.362,A -85,B 0,C 180,E1 -7180.089,E2 -7180.089} C_VEL
LIN {X 0,Y 474.611,Z 134.367,A -85,B 0,C 180,E1 -7182.773,E2 -7182.773} C_VEL
LIN {X 0,Y 474.623,Z 134.363,A -85,B 0,C 180,E1 -7185.42,E2 -7185.42} C_VEL
LIN {X 0,Y 474.692,Z 134.356,A -85,B 0,C 180,E1 -7188.037,E2 -7188.037} C_VEL
LIN {X 0,Y 474.695,Z 134.354,A -85,B 0,C 180,E1 -7191.486,E2 -7191.486} C_VEL
LIN {X 0,Y 474.725,Z 134.352,A -85,B 0,C 180,E1 -7194.052,E2 -7194.052} C_VEL
LIN {X 0,Y 474.859,Z 134.335,A -85,B 0,C 180,E1 -7197.455,E2 -7197.455} C_VEL
LIN {X 0,Y 474.866,Z 134.334,A -85,B 0,C 180,E1 -7200,E2 -7200} C_VEL
LIN {X 0,Y 474.86,Z 134.334,A -85,B 0,C 180,E1 -7202.545,E2 -7202.545} C_VEL
LIN {X 0,Y 474.731,Z 134.351,A -85,B 0,C 180,E1 -7205.948,E2 -7205.948} C_VEL
LIN {X 0,Y 474.695,Z 134.354,A -85,B 0,C 180,E1 -7208.514,E2 -7208.514} C_VEL
LIN {X 0,Y 474.692,Z 134.356,A -85,B 0,C 180,E1 -7211.963,E2 -7211.963} C_VEL
LIN {X 0,Y 474.667,Z 134.358,A -85,B 0,C 180,E1 -7215.767,E2 -7215.767} C_VEL
LIN {X 0,Y 474.649,Z 134.363,A -85,B 0,C 180,E1 -7219.011,E2 -7219.011} C_VEL
LIN {X 0,Y 474.576,Z 134.37,A -85,B 0,C 180,E1 -7221.73,E2 -7221.73} C_VEL
LIN {X 0,Y 474.615,Z 134.364,A -85,B 0,C 180,E1 -7224.495,E2 -7224.495} C_VEL
LIN {X 0,Y 474.663,Z 134.359,A -85,B 0,C 180,E1 -7227.333,E2 -7227.333} C_VEL
LIN {X 0,Y 474.594,Z 134.366,A -85,B 0,C 180,E1 -7230.231,E2 -7230.231} C_VEL
LIN {X 0,Y 474.615,Z 134.364,A -85,B 0,C 180,E1 -7233.222,E2 -7233.222} C_VEL
LIN {X 0,Y 474.579,Z 134.369,A -85,B 0,C 180,E1 -7236.324,E2 -7236.324} C_VEL
LIN {X 0,Y 474.609,Z 134.363,A -85,B 0,C 180,E1 -7239.647,E2 -7239.647} C_VEL
LIN {X 0,Y 474.616,Z 134.366,A -85,B 0,C 180,E1 -7242.238,E2 -7242.238} C_VEL
LIN {X 0,Y 474.61,Z 134.363,A -85,B 0,C 180,E1 -7245.299,E2 -7245.299} C_VEL
LIN {X 0,Y 474.614,Z 134.368,A -85,B 0,C 180,E1 -7248.216,E2 -7248.216} C_VEL
LIN {X 0,Y 474.639,Z 134.363,A -85,B 0,C 180,E1 -7250.455,E2 -7250.455} C_VEL
LIN {X 0,Y 474.584,Z 134.367,A -85,B 0,C 180,E1 -7253.678,E2 -7253.678} C_VEL
LIN {X 0,Y 474.639,Z 134.359,A -85,B 0,C 180,E1 -7256.781,E2 -7256.781} C_VEL
LIN {X 0,Y 474.602,Z 134.367,A -85,B 0,C 180,E1 -7259.771,E2 -7259.771} C_VEL
LIN {X 0,Y 474.695,Z 134.353,A -85,B 0,C 180,E1 -7262.681,E2 -7262.681} C_VEL
LIN {X 0,Y 474.693,Z 134.451,A -85,B 0,C 180,E1 -7263.912,E2 -7263.912} C_VEL
LIN {X 0,Y 476.728,Z 145.591,A -85,B 0,C 180,E1 -7265.901,E2 -7265.901} C_VEL
LIN {X 0,Y 476.183,Z 161.322,A -85,B 0,C 180,E1 -7268.518,E2 -7268.518} C_VEL
LIN {X 0,Y 475.516,Z 180.666,A -85,B 0,C 180,E1 -7271.696,E2 -7271.696} C_VEL
LIN {X 0,Y 475.204,Z 190.546,A -85,B 0,C 180,E1 -7273.301,E2 -7273.301} C_VEL
LIN {X 0,Y 477.876,Z 209.973,A -85,B 0,C 180,E1 -7273.684,E2 -7273.684} C_VEL
LIN {X 0,Y 477.274,Z 299.088,A -85,B 0,C 180,E1 -7275.041,E2 -7275.041} C_VEL
LIN {X 0,Y 476.933,Z 311.652,A -85,B 0,C 180,E1 -7275.384,E2 -7275.384} C_VEL
LIN {X 0,Y 476.461,Z 324.625,A -85,B 0,C 180,E1 -7275.915,E2 -7275.915} C_VEL
LIN {X 0,Y 476.03,Z 336.129,A -85,B 0,C 180,E1 -7276.555,E2 -7276.555} C_VEL
LIN {X 0,Y 475.553,Z 348.037,A -85,B 0,C 180,E1 -7277.419,E2 -7277.419} C_VEL
LIN {X 0,Y 475.111,Z 358.528,A -85,B 0,C 180,E1 -7278.374,E2 -7278.374} C_VEL
LIN {X 0,Y 474.716,Z 367.184,A -85,B 0,C 180,E1 -7279.336,E2 -7279.336} C_VEL
LIN {X 0,Y 474.391,Z 375.164,A -85,B 0,C 180,E1 -7280.407,E2 -7280.407} C_VEL
LIN {X 0,Y 474.104,Z 382.966,A -85,B 0,C 180,E1 -7281.691,E2 -7281.691} C_VEL
LIN {X 0,Y 473.894,Z 390.133,A -85,B 0,C 180,E1 -7283.187,E2 -7283.187} C_VEL
LIN {X 0,Y 473.835,Z 394.909,A -85,B 0,C 180,E1 -7284.468,E2 -7284.468} C_VEL
LIN {X 0,Y 473.735,Z 398.556,A -85,B 0,C 180,E1 -7285.747,E2 -7285.747} C_VEL
LIN {X 0,Y 473.823,Z 400.447,A -85,B 0,C 180,E1 -7286.599,E2 -7286.599} C_VEL
LIN {X 0,Y 473.765,Z 401.861,A -85,B 0,C 180,E1 -7287.45,E2 -7287.45} C_VEL
LIN {X 0,Y 473.757,Z 402.869,A -85,B 0,C 180,E1 -7288.301,E2 -7288.301} C_VEL
LIN {X 0,Y 473.682,Z 403.711,A -85,B 0,C 180,E1 -7290.001,E2 -7290.001} C_VEL
LIN {X 0,Y 473.757,Z 402.906,A -85,B 0,C 180,E1 -7291.701,E2 -7291.701} C_VEL
LIN {X 0,Y 473.806,Z 400.525,A -85,B 0,C 180,E1 -7293.402,E2 -7293.402} C_VEL
LIN {X 0,Y 473.76,Z 397.59,A -85,B 0,C 180,E1 -7294.681,E2 -7294.681} C_VEL
LIN {X 0,Y 473.803,Z 393.624,A -85,B 0,C 180,E1 -7295.961,E2 -7295.961} C_VEL
LIN {X 0,Y 474,Z 387.542,A -85,B 0,C 180,E1 -7297.455,E2 -7297.455} C_VEL
LIN {X 0,Y 474.202,Z 380.888,A -85,B 0,C 180,E1 -7298.738,E2 -7298.738} C_VEL
LIN {X 0,Y 474.507,Z 372.638,A -85,B 0,C 180,E1 -7300.023,E2 -7300.023} C_VEL
LIN {X 0,Y 474.983,Z 364.214,A -85,B 0,C 180,E1 -7301.091,E2 -7301.091} C_VEL
LIN {X 0,Y 475.37,Z 354.251,A -85,B 0,C 180,E1 -7302.124,E2 -7302.124} C_VEL
LIN {X 0,Y 475.811,Z 343.577,A -85,B 0,C 180,E1 -7303.018,E2 -7303.018} C_VEL
LIN {X 0,Y 476.308,Z 332.38,A -85,B 0,C 180,E1 -7303.765,E2 -7303.765} C_VEL
LIN {X 0,Y 476.804,Z 319.845,A -85,B 0,C 180,E1 -7304.403,E2 -7304.403} C_VEL
LIN {X 0,Y 477.251,Z 307.356,A -85,B 0,C 180,E1 -7304.853,E2 -7304.853} C_VEL
LIN {X 0,Y 477.542,Z 294.755,A -85,B 0,C 180,E1 -7305.143,E2 -7305.143} C_VEL
LIN {X 0,Y 478.117,Z 209.26,A -85,B 0,C 180,E1 -7306.443,E2 -7306.443} C_VEL
LIN {X 0,Y 475.274,Z 190.22,A -85,B 0,C 180,E1 -7306.871,E2 -7306.871} C_VEL
LIN {X 0,Y 475.864,Z 173.635,A -85,B 0,C 180,E1 -7309.611,E2 -7309.611} C_VEL
LIN {X 0,Y 476.622,Z 156.093,A -85,B 0,C 180,E1 -7312.544,E2 -7312.544} C_VEL
LIN {X 0,Y 477.015,Z 146.788,A -85,B 0,C 180,E1 -7314.12,E2 -7314.12} C_VEL
LIN {X 0,Y 475.209,Z 136.95,A -85,B 0,C 180,E1 -7315.925,E2 -7315.925} C_VEL
LIN {X 0,Y 474.661,Z 134.361,A -85,B 0,C 180,E1 -7316.431,E2 -7316.431} C_VEL
LIN {X 0,Y 474.61,Z 134.368,A -85,B 0,C 180,E1 -7319.253,E2 -7319.253} C_VEL
LIN {X 0,Y 474.618,Z 134.366,A -85,B 0,C 180,E1 -7322.431,E2 -7322.431} C_VEL
LIN {X 0,Y 474.614,Z 134.365,A -85,B 0,C 180,E1 -7325.469,E2 -7325.469} C_VEL
LIN {X 0,Y 474.612,Z 134.361,A -85,B 0,C 180,E1 -7328.458,E2 -7328.458} C_VEL
LIN {X 0,Y 474.617,Z 134.365,A -85,B 0,C 180,E1 -7331.786,E2 -7331.786} C_VEL
LIN {X 0,Y 474.618,Z 134.367,A -85,B 0,C 180,E1 -7335.298,E2 -7335.298} C_VEL
LIN {X 0,Y 474.61,Z 134.362,A -85,B 0,C 180,E1 -7338.213,E2 -7338.213} C_VEL
LIN {X 0,Y 474.61,Z 134.366,A -85,B 0,C 180,E1 -7341.542,E2 -7341.542} C_VEL
LIN {X 0,Y 474.622,Z 134.364,A -85,B 0,C 180,E1 -7344.725,E2 -7344.725} C_VEL
LIN {X 0,Y 474.633,Z 134.36,A -85,B 0,C 180,E1 -7347.787,E2 -7347.787} C_VEL
LIN {X 0,Y 474.598,Z 134.371,A -85,B 0,C 180,E1 -7350.89,E2 -7350.89} C_VEL
LIN {X 0,Y 474.59,Z 134.364,A -85,B 0,C 180,E1 -7353.624,E2 -7353.624} C_VEL
LIN {X 0,Y 474.633,Z 134.365,A -85,B 0,C 180,E1 -7356.642,E2 -7356.642} C_VEL
LIN {X 0,Y 474.641,Z 134.357,A -85,B 0,C 180,E1 -7360.089,E2 -7360.089} C_VEL
LIN {X 0,Y 474.592,Z 134.368,A -85,B 0,C 180,E1 -7362.772,E2 -7362.772} C_VEL
LIN {X 0,Y 474.625,Z 134.355,A -85,B 0,C 180,E1 -7365.42,E2 -7365.42} C_VEL
LIN {X 0,Y 474.683,Z 134.356,A -85,B 0,C 180,E1 -7368.037,E2 -7368.037} C_VEL
LIN {X 0,Y 474.659,Z 134.351,A -85,B 0,C 180,E1 -7371.485,E2 -7371.485} C_VEL
LIN {X 0,Y 474.733,Z 134.353,A -85,B 0,C 180,E1 -7374.052,E2 -7374.052} C_VEL
LIN {X 0,Y 474.868,Z 134.326,A -85,B 0,C 180,E1 -7377.455,E2 -7377.455} C_VEL
LIN {X 0,Y 474.878,Z 134.335,A -85,B 0,C 180,E1 -7380,E2 -7380} C_VEL
LIN {X 0,Y 474.87,Z 134.324,A -85,B 0,C 180,E1 -7382.545,E2 -7382.545} C_VEL
LIN {X 0,Y 474.735,Z 134.35,A -85,B 0,C 180,E1 -7385.948,E2 -7385.948} C_VEL
LIN {X 0,Y 474.703,Z 134.344,A -85,B 0,C 180,E1 -7388.514,E2 -7388.514} C_VEL
LIN {X 0,Y 474.704,Z 134.352,A -85,B 0,C 180,E1 -7391.963,E2 -7391.963} C_VEL
LIN {X 0,Y 474.68,Z 134.356,A -85,B 0,C 180,E1 -7395.767,E2 -7395.767} C_VEL
LIN {X 0,Y 474.662,Z 134.359,A -85,B 0,C 180,E1 -7399.011,E2 -7399.011} C_VEL
LIN {X 0,Y 474.588,Z 134.366,A -85,B 0,C 180,E1 -7401.729,E2 -7401.729} C_VEL
LIN {X 0,Y 474.627,Z 134.358,A -85,B 0,C 180,E1 -7404.495,E2 -7404.495} C_VEL
LIN {X 0,Y 474.638,Z 134.36,A -85,B 0,C 180,E1 -7407.324,E2 -7407.324} C_VEL
LIN {X 0,Y 474.602,Z 134.363,A -85,B 0,C 180,E1 -7410.231,E2 -7410.231} C_VEL
LIN {X 0,Y 474.626,Z 134.361,A -85,B 0,C 180,E1 -7413.222,E2 -7413.222} C_VEL
LIN {X 0,Y 474.59,Z 134.367,A -85,B 0,C 180,E1 -7416.324,E2 -7416.324} C_VEL
